// ---- GlobalTextList.TcGTLO
TEXTLIST GlobalTextList
  3955 = ' %5.2f h'
  1376 = ' %d %%'
  307 = ' %d days'
  1111 = '%2.1f  mA'
  102 = '%5.1f W'
  269 = '%5.2f h'
  621 = '%d'
  1617 = '%d %%'
  2081 = '%d days'
  3200 = '%d h'
  1372 = '%d Hz'
  2105 = '%d min'
  2025 = '%d ms'
  1540 = '%d s'
  1613 = '%d V'
  2272 = '%d weeks'
  1359 = '%d °C'
  376 = '%s'
  640 = '0'
  641 = '1'
  661 = '10'
  662 = '11'
  663 = '12'
  999 = '13'
  1000 = '14'
  1001 = '15'
  1002 = '16'
  1003 = '17'
  1004 = '18'
  1005 = '19'
  195 = '2'
  1006 = '20'
  1007 = '21'
  1008 = '22'
  1009 = '23'
  1010 = '24'
  1011 = '25'
  1012 = '26'
  1013 = '27'
  1014 = '28'
  1015 = '29'
  654 = '3'
  1016 = '30'
  1017 = '31'
  1018 = '32'
  1019 = '33'
  1020 = '34'
  1021 = '35'
  1022 = '36'
  1023 = '37'
  1024 = '38'
  1025 = '39'
  655 = '4'
  1026 = '40'
  1027 = '41'
  1028 = '42'
  1029 = '43'
  1030 = '44'
  1031 = '45'
  1032 = '46'
  1033 = '47'
  1034 = '48'
  1035 = '49'
  656 = '5'
  358 = '50'
  359 = '51'
  360 = '52'
  361 = '53'
  362 = '54'
  363 = '55'
  364 = '56'
  365 = '57'
  366 = '58'
  367 = '59'
  657 = '6'
  368 = '60'
  369 = '61'
  370 = '62'
  371 = '63'
  658 = '7'
  659 = '8'
  660 = '9'
  1089 = 'AC-supply possible'
  644 = 'Actual Level:'
  650 = 'Address Type'
  236 = 'Addressing Per Physical Selection Supported'
  1533 = 'Adjustable Emergency Level'
  1175 = 'AM Operation active:'
  1044 = 'AM operation possible'
  1045 = 'Auto Test Capability'
  1799 = 'Battery Charge'
  710 = 'Battery Duration Failure'
  3347 = 'Battery Failure'
  3316 = 'Battery Fully Charged'
  2471 = 'Bit 0'
  379 = 'Bit 1'
  2734 = 'Bit 2'
  2320 = 'Bit 3'
  929 = 'Bit 4'
  2576 = 'Bit 5'
  2065 = 'Bit 6'
  1623 = 'Bit 7'
  6 = 'Bottom Button'
  728 = 'Broadcast'
  482 = 'Button 1'
  720 = 'Button 2'
  515 = 'Button pressed'
  498 = 'Button released'
  527 = 'Button stuck / free'
  3304 = 'Cancel Hold Timer'
  2101 = 'Catch Movement'
  2319 = 'Catching:'
  897 = 'Change Addresses'
  1971 = 'Checkbox'
  372 = 'Choose group:'
  98 = 'Choose scene:'
  1571 = 'Circuit Failure'
  672 = 'Commands'
  618 = 'Complete new installation \n(all addresses will be removed)'
  807 = 'Control'
  645 = 'Control Gear Failure:'
  445 = 'Current protection active:'
  1716 = 'Current protection device'
  668 = 'Current protection enabled:'
  5 = 'Current Protector Enabled '
  1902 = 'DALI Line:'
  1135 = 'DC-supply possible'
  560 = 'Deadtime Timer:'
  1180 = 'DI1 falling edge'
  1218 = 'DI1 rising edge'
  1726 = 'DI2 falling edge'
  1876 = 'DI2 rising edge'
  519 = 'Dim Dwn'
  63 = 'Dim Up'
  2002 = 'Dimmer Temperature'
  936 = 'Dimming Curve:'
  1317 = 'Dimming method bit 0'
  776 = 'Dimming method bit 1'
  2135 = 'Do not lock process image in case of \nDALI commands from DI1 or DI2'
  4011 = 'Double press'
  1112 = 'Double Timer Min:'
  3936 = 'Double Timer:'
  811 = 'Down'
  594 = 'Down Switch-Off Threshold'
  2357 = 'Down Switch-On Threshold'
  1482 = 'Duration Test Delay Time'
  3527 = 'Duration Test Done And Result Valid'
  3086 = 'Duration Test Failed'
  3077 = 'Duration Test Interval'
  2631 = 'Duration Test Is In Progress'
  2791 = 'Duration Test Max. Delay Exceed'
  1708 = 'Duration Test Request Pending'
  2905 = 'Duration Test Result'
  1759 = 'Emergency Lamp Failure'
  779 = 'Emergency Level'
  3733 = 'Emergency MaxLevel'
  3168 = 'Emergency Min Level'
  1204 = 'Emergency Mode'
  971 = 'Emergency Mode Active'
  1901 = 'Emergency Status'
  486 = 'Enable'
  828 = 'Enable:'
  1982 = 'EventPriority'
  32 = 'EventPriority:'
  494 = 'EventScheme'
  1113 = 'EventScheme:'
  125 = 'Extended Emergency Mode Active'
  1841 = 'Extended Fade Time only valid if Fade Time equals 0!'
  3956 = 'Extended Version'
  649 = 'Fade Running:'
  1345 = 'FadeRate'
  1352 = 'FadeTime'
  1610 = 'Failure Status'
  319 = 'Fast Fade Time:'
  2099 = 'Features'
  425 = 'Features (Read only)'
  206 = 'Features Byte 1'
  377 = 'Features Byte 2'
  2876 = 'Features Byte 3'
  3334 = 'Function Test Delay Time'
  3242 = 'Function Test Done And Result Valid'
  2712 = 'Function Test Failed'
  1801 = 'Function Test Interval'
  1945 = 'Function Test Is In Progress'
  3448 = 'Function Test Max. Delay Exceed'
  165 = 'Function Test Request Pending'
  967 = 'Gang 1.312A'
  256 = 'Gang 1.315'
  906 = 'Gang 1.316'
  207 = 'Gang 2.344'
  66 = 'Gang 2.344A'
  406 = 'Gang 4.308'
  524 = 'Gang 6.310'
  316 = 'Gang 7.301'
  3204 = 'Gear Type'
  1989 = 'GearType'
  815 = 'Go to Scene'
  99 = 'Go to scene'
  721 = 'Group Address'
  2361 = 'Hardwired Inhibit Is Active'
  3553 = 'Hardwired Inhibit Supported'
  2225 = 'Hardwired Switch Is On'
  568 = 'Hold Timer:'
  199 = 'Hysteresis Min:'
  200 = 'Hysteresis:'
  790 = 'Identification Active'
  315 = 'Illuminance Level'
  37 = 'Inhibit'
  3340 = 'Inhibit Mode'
  540 = 'Input Value:'
  544 = 'Instance Error:'
  1038 = 'Instance Number:'
  3047 = 'Integral Control Gear'
  492 = 'Internal DALI power supply disabled'
  1771 = 'K-Bus Watchdog'
  3636 = 'Lamp Emergency Time'
  647 = 'Lamp Failure:'
  2812 = 'Lamp Total Operation Time'
  1521 = 'Leading Edge Mode Running'
  506 = 'LED module integrated'
  2077 = 'Linear Dimming Curve Active'
  2179 = 'Load current can be queried '
  1266 = 'Load Current Overload'
  1355 = 'Load current overload with output \nlevel reduction can be queried'
  306 = 'Load Decrease:'
  1137 = 'Load Increase:'
  2313 = 'Load over-current can be queried'
  2518 = 'Load Over-Current Shutdown'
  1226 = 'Load Rating'
  2963 = 'Load rating can be queried'
  2785 = 'Load unsuitable can be queried'
  1454 = 'Load voltage can be queried'
  516 = 'Load Voltage Out Of Limits'
  1811 = 'Lockable bytes: changeable if "Offset 2" has the Value 85 (0x55).\nFor changing use decimal value.'
  523 = 'Long press repeat'
  507 = 'Long press start'
  511 = 'Long press stop'
  43 = 'Lys Auto'
  444 = 'Lys Rum'
  489 = 'Lys Zone 1'
  2032 = 'Maintained Control Gear'
  2046 = 'Memory Bank:'
  3290 = 'Movement'
  531 = 'na'
  23 = 'Name'
  926 = 'Name of byte in memory bank'
  1417 = 'NewAddress'
  588 = 'No Movement'
  1061 = 'Non-logarithmic dimming curve can \nbe selected'
  1795 = 'Normal Mode Active'
  572 = 'Occupied'
  808 = 'Off'
  22 = 'Offset'
  1329 = 'Offset in memory bank'
  1409 = 'OldAddress'
  816 = 'On and Step Up'
  1207 = 'Open circuit detection can be queried'
  277 = 'Open Circuit:'
  1375 = 'Open Ciruit (No Load) Detect'
  619 = 'Optical feedback'
  963 = 'Output is current controlled'
  844 = 'Output regulated by current:'
  676 = 'Parameters'
  2547 = 'Parameters Absolute Input Device'
  1580 = 'Parameters Generic Instance'
  2259 = 'Parameters LED'
  309 = 'Parameters Light Sensor'
  556 = 'Parameters Occupancy Sensor'
  465 = 'Parameters Pushbutton Sensor'
  3234 = 'Physical Selection Supported'
  1847 = 'Physical selection supported'
  708 = 'PIR'
  457 = 'PIR status'
  1071 = 'Please check if Current Protector is present \nby reading parameters first.'
  308 = 'Please select the desired Short Address in the table above.'
  1458 = 'Please select the function you need from dropdown above'
  751 = 'Position Event'
  245 = 'Possible Operating Modes'
  719 = 'Power pulse operation'
  1744 = 'Power supply integrated'
  1561 = 'PP Operation active:'
  2321 = 'Prolong Time (30sec / Step)'
  970 = 'PWM Operation active:'
  1882 = 'PWM operation possible'
  1487 = 'Query idle time detection \nenabled'
  701 = 'Query load decrease enabled'
  1351 = 'Query load increase enabled'
  837 = 'Query reduction luminous flux \nregarding thermal overload'
  463 = 'Query short circuit enabled'
  1293 = 'Query thermal switch enabled'
  617 = 'Random Addressing'
  2174 = 'Rated Duration'
  881 = 'Re-Light / Reset Inhibit'
  373 = 'Read'
  1611 = 'Read Only'
  1531 = 'Reads all Fading Parameters'
  768 = 'Real Load Power'
  854 = 'Real load power can be queried'
  810 = 'Recall Max Level'
  809 = 'Recall Min Level'
  186 = 'Ref. Measurement failed:'
  439 = 'Reference System Power'
  2713 = 'Relight Rest Mode Supported'
  580 = 'Repeat'
  470 = 'Repeat Timer:'
  1913 = 'Report Timer:'
  716 = 'Reset Duration Test Done Flag'
  592 = 'Reset Function Test Done Flag'
  2418 = 'Reset inactive process image'
  3150 = 'Reset Lamp Time'
  648 = 'Reset State:'
  1037 = 'Resolution:'
  299 = 'Rest'
  591 = 'Rest Mode Active'
  2001 = 'RMS Load Current'
  784 = 'RMS Load Voltage'
  586 = 'RMS Supply Voltage'
  874 = 'Rum 1.106'
  65 = 'Rum 1.108'
  175 = 'Rum 1.111A'
  924 = 'Rum 1.111C'
  219 = 'Rum 1.111D'
  690 = 'Rum 1.111E'
  912 = 'Rum 1.115'
  126 = 'Rum 1.118'
  215 = 'Rum 1.312A'
  725 = 'Rum 1.318'
  839 = 'Rum 1.319'
  456 = 'Rum 1.320'
  800 = 'Rum 1.321'
  622 = 'Rum 1.322'
  646 = 'Rum 1.323'
  966 = 'Rum 1.324'
  95 = 'Rum 1.325'
  335 = 'Rum 1.326'
  150 = 'Rum 1.327'
  651 = 'Rum 1.328'
  980 = 'Rum 1.330'
  262 = 'Rum 1115'
  642 = 'Rum 2.341'
  978 = 'Rum 2.345'
  736 = 'Rum 2.349'
  430 = 'Rum 6.310 Sofagruppe'
  348 = 'Rum 6.327'
  891 = 'Rum 6.328'
  11 = 'Rum 6.329'
  72 = 'Rum 6.330B'
  197 = 'Rum 6.331'
  564 = 'Rum 6.333'
  997 = 'Rum 6.337'
  31 = 'Rum 6_330A'
  616 = 'Scan devices by address'
  1036 = 'Scene Level'
  814 = 'Scene:'
  1366 = 'Set Extended Fade Time'
  252 = 'Set Fade Rate'
  1875 = 'Set Fade Time'
  715 = 'Short Address'
  1367 = 'Short Address Range'
  1041 = 'Short Address:'
  34 = 'Short Circuit:'
  503 = 'Short press'
  1516 = 'Short Timer Min:'
  478 = 'Short Timer:'
  2548 = 'Shutdown Invalid Dimming Method'
  1360 = 'Single Short Address'
  395 = 'SP_Lux: %.0f'
  525 = 'SP_Lux: %f'
  615 = 'Start'
  582 = 'Start Duration Test'
  2374 = 'Start Function Test'
  155 = 'Start Identification'
  620 = 'Start with address:'
  2346 = 'State Incandescent Lamp'
  643 = 'Status'
  958 = 'Status Absolute Input Device'
  2506 = 'Status Generic Instance'
  2252 = 'Status LED'
  317 = 'Status Light Sensor'
  597 = 'Status Occupancy Sensor'
  536 = 'Status Pushbutton Sensor'
  558 = 'Step Down'
  813 = 'Step Down and Off'
  818 = 'Step Up'
  1193 = 'Stop Test'
  164 = 'Stuck Timer:'
  1256 = 'Supply Frequency'
  2271 = 'Supply frequency can be queried'
  1975 = 'Supply Frequency Out of Limits'
  2505 = 'Supply voltage can be queried'
  2707 = 'Supply Voltage Out Of Limits'
  1042 = 'Switch Off'
  375 = 'Switch On'
  3781 = 'Switched Maintained Control Gear'
  2168 = 'Temperature can be queried'
  2458 = 'Terminal Event'
  1848 = 'Test Execution Timeout'
  849 = 'Test Type A'
  2013 = 'Thermal Overload'
  2042 = 'Thermal Overload with output\nlevel reduction can be queried'
  1108 = 'Thermal Overload:'
  355 = 'Thermal Shut Down:'
  2507 = 'Thermal Shutdown'
  2226 = 'Thermal Shutdown can be queried'
  2733 = 'Threshold Editable'
  305 = 'To'
  973 = 'Top Button'
  136 = 'Trailing Edge ModeRunning'
  734 = 'Unaddressed'
  817 = 'Up'
  3123 = 'Up Switch-Off Threshold'
  1449 = 'Up Switch-On Threshold'
  2521 = 'V%s'
  576 = 'Vacant'
  1205 = 'Value'
  24 = 'Value Dec'
  1435 = 'Value decimal'
  25 = 'Value Hex'
  2231 = 'Value hexadecimal,\nto change use\nvalue decimal'
  374 = 'Write'
  2104 = 'Write\nDimming Curve'
  1047 = 'Write default values'
  490 = 'Write parameters'
END_TEXTLIST

// ---- POUs/Alle_Rum/Gange/Gang_1_316/Visualization_1_316.TcVIS
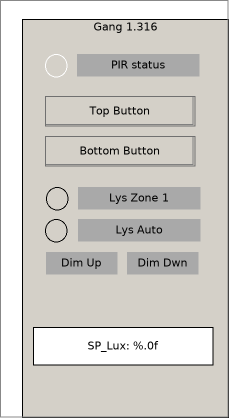
VISUALIZATION Visualization_1_316  // 229x418
    RoundedRectangle (22,19 207x399), "Gang 1.316"
    Rectangle (33,327 180x38), "SP_Lux: %.0f", text variable: P_Gang_1_316.fbLys.fbLightCtrl.fLuxZone1
    Button (45,96 150x30), "Top Button"
        tap P_Gang_1_316.bButtonZone1_Visu
    Button (45,136 150x30), "Bottom Button"
        tap P_Gang_1_316.bBottomButtonZone1_Visu
    Ellipse (46,187 22x23), colour toggle: P_Gang_1_316.fbLys.fbLightCtrl.bOnZone1
    Rectangle (78,187 122x22), "Lys Zone 1"
    Rectangle (46,252 71x22), "Dim Up", colour toggle: P_Gang_1_316.fbLys.fbLightCtrl.bDimUp
    Rectangle (127,252 71x22), "Dim Dwn", colour toggle: P_Gang_1_316.fbLys.fbLightCtrl.bDimDwn
    Ellipse (45,219 22x23), colour toggle: P_Gang_1_316.fbLys.fbLightCtrl.bAutoZone1
    Rectangle (78,219 122x22), "Lys Auto"
    Ellipse (45,54 22x23), colour toggle: P_Gang_1_316.fbLys.fbLightCtrl.bPIR
    Rectangle (77,54 122x22), "PIR status"
END_VISUALIZATION

// ---- POUs/Alle_Rum/Gange/Gang_7_301_en_linje_en_pendel_1/Visualization_4_308_1_1.TcVIS
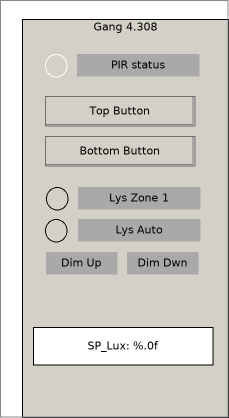
VISUALIZATION Visualization_4_308_1_1  // 229x418
    RoundedRectangle (22,19 207x399), "Gang 4.308"
    Rectangle (33,327 180x38), "SP_Lux: %.0f", text variable: P_Gang_4_308.arrfbLysGruppe[1].fbLightCtrl.fLuxZone1
    Button (45,96 150x30), "Top Button"
        tap P_Gang_4_308.bButtonZone1_Visu
    Button (45,136 150x30), "Bottom Button"
        tap P_Gang_4_308.bBottomButtonZone1_Visu
    Ellipse (46,187 22x23), colour toggle: P_Gang_4_308.fbLys.fbLightCtrl.bOnZone1
    Rectangle (78,187 122x22), "Lys Zone 1"
    Rectangle (46,252 71x22), "Dim Up", colour toggle: P_Gang_4_308.arrfbLysGruppe[1].fbLightCtrl.bDimUp
    Rectangle (127,252 71x22), "Dim Dwn", colour toggle: P_Gang_4_308.arrfbLysGruppe[1].fbLightCtrl.bDimDwn
    Ellipse (45,219 22x23), colour toggle: P_Gang_4_308.arrfbLysGruppe[1].fbLightCtrl.bAutoZone1
    Rectangle (78,219 122x22), "Lys Auto"
    Ellipse (45,54 22x23), colour toggle: P_Gang_4_308.arrfbLysGruppe[1].fbLightCtrl.bPIR
    Rectangle (77,54 122x22), "PIR status"
END_VISUALIZATION

// ---- POUs/Alle_Rum/Gange/Gang_2_346A/Visualization_2_346A.TcVIS
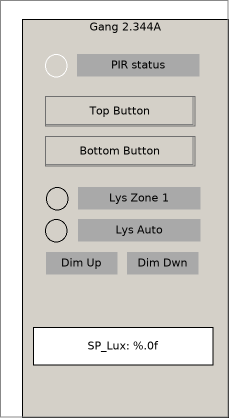
VISUALIZATION Visualization_2_346A  // 229x418
    RoundedRectangle (22,19 207x399), "Gang 2.344A"
    Rectangle (33,327 180x38), "SP_Lux: %.0f", text variable: P_Gang_2_346A.fbLys.fbLightCtrl.fLuxZone1
    Button (45,96 150x30), "Top Button"
        tap P_Gang_2_346A.bTopButtonZone1_Visu
    Button (45,136 150x30), "Bottom Button"
        tap P_Gang_2_346A.bBottomButtonZone1_Visu
    Ellipse (46,187 22x23), colour toggle: P_Gang_2_346A.fbLys.fbLightCtrl.bOnZone1
    Rectangle (78,187 122x22), "Lys Zone 1"
    Rectangle (46,252 71x22), "Dim Up", colour toggle: P_Gang_2_346A.fbLys.fbLightCtrl.bDimUp
    Rectangle (127,252 71x22), "Dim Dwn", colour toggle: P_Gang_2_346A.fbLys.fbLightCtrl.bDimDwn
    Ellipse (45,219 22x23), colour toggle: P_Gang_2_346A.fbLys.fbLightCtrl.bAutoZone1
    Rectangle (78,219 122x22), "Lys Auto"
    Ellipse (45,54 22x23), colour toggle: P_Gang_2_346A.fbLys.fbLightCtrl.bPIR
    Rectangle (77,54 122x22), "PIR status"
END_VISUALIZATION

// ---- POUs/Alle_Rum/Gange/Gang_2_344/Visualization_4_308_1_1_1.TcVIS
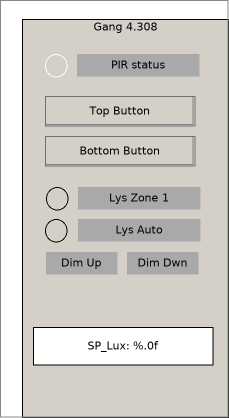
VISUALIZATION Visualization_4_308_1_1_1  // 229x418
    RoundedRectangle (22,19 207x399), "Gang 4.308"
    Rectangle (33,327 180x38), "SP_Lux: %.0f", text variable: P_Gang_4_308.arrfbLysGruppe[1].fbLightCtrl.fLuxZone1
    Button (45,96 150x30), "Top Button"
        tap P_Gang_4_308.bButtonZone1_Visu
    Button (45,136 150x30), "Bottom Button"
        tap P_Gang_4_308.bBottomButtonZone1_Visu
    Ellipse (46,187 22x23), colour toggle: P_Gang_4_308.fbLys.fbLightCtrl.bOnZone1
    Rectangle (78,187 122x22), "Lys Zone 1"
    Rectangle (46,252 71x22), "Dim Up", colour toggle: P_Gang_4_308.arrfbLysGruppe[1].fbLightCtrl.bDimUp
    Rectangle (127,252 71x22), "Dim Dwn", colour toggle: P_Gang_4_308.arrfbLysGruppe[1].fbLightCtrl.bDimDwn
    Ellipse (45,219 22x23), colour toggle: P_Gang_4_308.arrfbLysGruppe[1].fbLightCtrl.bAutoZone1
    Rectangle (78,219 122x22), "Lys Auto"
    Ellipse (45,54 22x23), colour toggle: P_Gang_4_308.arrfbLysGruppe[1].fbLightCtrl.bPIR
    Rectangle (77,54 122x22), "PIR status"
END_VISUALIZATION

// ---- POUs/Alle_Rum/Rum_Med_DALI_Pir/Rum_2_341/Visualization_2_341.TcVIS
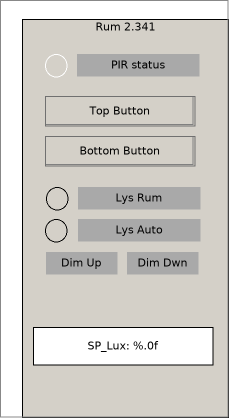
VISUALIZATION Visualization_2_341  // 229x418
    RoundedRectangle (22,19 207x399), "Rum 2.341"
    Rectangle (33,327 180x38), "SP_Lux: %.0f", text variable: P_Rum_2_341.fbLys.fbLightCtrl.fLuxZone1
    Button (45,96 150x30), "Top Button"
        tap P_Rum_2_341.bTopButtonZone1_Visu
    Button (45,136 150x30), "Bottom Button"
        tap P_Rum_2_341.bBottomButtonZone1_Visu
    Ellipse (46,187 22x23), colour toggle: P_Rum_2_341.fbLys.fbLightCtrl.bOnZone1
    Rectangle (78,187 122x22), "Lys Rum"
    Rectangle (46,252 71x22), "Dim Up", colour toggle: P_Rum_2_341.fbLys.fbLightCtrl.bDimUp
    Rectangle (127,252 71x22), "Dim Dwn", colour toggle: P_Rum_2_341.fbLys.fbLightCtrl.bDimDwn
    Ellipse (45,219 22x23), colour toggle: P_Rum_2_341.fbLys.fbLightCtrl.bAutoZone1
    Rectangle (78,219 122x22), "Lys Auto"
    Ellipse (45,54 22x23), colour toggle: P_Rum_2_341.fbLys.fbLightCtrl.bPIR
    Rectangle (77,54 122x22), "PIR status"
END_VISUALIZATION

// ---- POUs/Alle_Rum/Rum_Med_DALI_Pir/Rum_2_345/Visualization_2_345.TcVIS
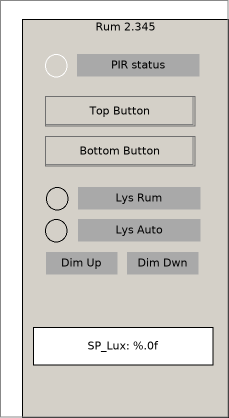
VISUALIZATION Visualization_2_345  // 229x418
    RoundedRectangle (22,19 207x399), "Rum 2.345"
    Rectangle (33,327 180x38), "SP_Lux: %.0f", text variable: P_Rum_2_345.fbLys.fbLightCtrl.fLuxZone1
    Button (45,96 150x30), "Top Button"
        tap P_Rum_2_345.bTopButtonZone1_Visu
    Button (45,136 150x30), "Bottom Button"
        tap P_Rum_2_345.bBottomButtonZone1_Visu
    Ellipse (46,187 22x23), colour toggle: P_Rum_2_345.fbLys.fbLightCtrl.bOnZone1
    Rectangle (78,187 122x22), "Lys Rum"
    Rectangle (46,252 71x22), "Dim Up", colour toggle: P_Rum_2_345.fbLys.fbLightCtrl.bDimUp
    Rectangle (127,252 71x22), "Dim Dwn", colour toggle: P_Rum_2_345.fbLys.fbLightCtrl.bDimDwn
    Ellipse (45,219 22x23), colour toggle: P_Rum_2_345.fbLys.fbLightCtrl.bAutoZone1
    Rectangle (78,219 122x22), "Lys Auto"
    Ellipse (45,54 22x23), colour toggle: P_Rum_2_345.fbLys.fbLightCtrl.bPIR
    Rectangle (77,54 122x22), "PIR status"
END_VISUALIZATION

// ---- POUs/Alle_Rum/Rum_Med_DALI_Pir/Rum_2_349/Visualization_2_349.TcVIS
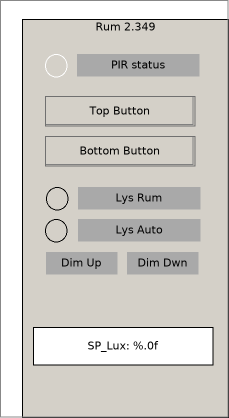
VISUALIZATION Visualization_2_349  // 229x418
    RoundedRectangle (22,19 207x399), "Rum 2.349"
    Rectangle (33,327 180x38), "SP_Lux: %.0f", text variable: P_Rum_2_349.fbLys.fbLightCtrl.fLuxZone1
    Button (45,96 150x30), "Top Button"
        tap P_Rum_2_349.bTopButtonZone1_Visu
    Button (45,136 150x30), "Bottom Button"
        tap P_Rum_2_349.bBottomButtonZone1_Visu
    Ellipse (46,187 22x23), colour toggle: P_Rum_2_349.fbLys.fbLightCtrl.bOnZone1
    Rectangle (78,187 122x22), "Lys Rum"
    Rectangle (46,252 71x22), "Dim Up", colour toggle: P_Rum_2_349.fbLys.fbLightCtrl.bDimUp
    Rectangle (127,252 71x22), "Dim Dwn", colour toggle: P_Rum_2_349.fbLys.fbLightCtrl.bDimDwn
    Ellipse (45,219 22x23), colour toggle: P_Rum_2_349.fbLys.fbLightCtrl.bAutoZone1
    Rectangle (78,219 122x22), "Lys Auto"
    Ellipse (45,54 22x23), colour toggle: P_Rum_2_349.fbLys.fbLightCtrl.bPIR
    Rectangle (77,54 122x22), "PIR status"
END_VISUALIZATION

// ---- POUs/DALI/DALI_Setup/VISUs/TextLists/CommandOnTerminalEvent.TcTLO
TEXTLIST CommandOnTerminalEvent
  0 = 'Do Nothing'
  1 = 'Off'
  2 = 'RecallMaxLevel'
  3 = 'RecallMinLevel'
  4 = 'GoToScene0'
  5 = 'GoToScene1'
  6 = 'GoToScene2'
  7 = 'GoToScene3'
  8 = 'GoToScene4'
  9 = 'GoToScene5'
  10 = 'GoToScene6'
  11 = 'GoToScene7'
  12 = 'GoToScene8'
  13 = 'GoToScene9'
  14 = 'GoToScene10'
  15 = 'GoToScene11'
  16 = 'GoToScene12'
  17 = 'GoToScene13'
  18 = 'GoToScene14'
  19 = 'GoToScene15'
   = ''
END_TEXTLIST

// ---- POUs/DALI/DALI_Setup/VISUs/TextLists/DimmingCurve.TcTLO
TEXTLIST DimmingCurve
  0 = 'Standard'
  1 = 'Linear'
  255 = 'Unknown'
   = ''
END_TEXTLIST

// ---- POUs/DALI/DALI_Setup/VISUs/TextLists/EventPriority.TcTLO
TEXTLIST EventPriority
  2 = 'MiddleHigh'
  3 = 'Middle'
  4 = 'MiddleLow'
  5 = 'Low'
  255 = 'Unknown'
   = ''
END_TEXTLIST

// ---- POUs/DALI/DALI_Setup/VISUs/TextLists/EventScheme.TcTLO
TEXTLIST EventScheme
  0 = '0 - Instance type and number'
  1 = '1 - Short address and instance type'
  2 = '2 - Short address and instance number'
  3 = '3 - Device group and instance type'
  4 = '4 - Instance group and instance type'
   = ''
END_TEXTLIST

// ---- POUs/DALI/DALI_Setup/VISUs/TextLists/ExtendedFadeTime.TcTLO
TEXTLIST ExtendedFadeTime
  0 = 'No Fade'
  1 = '1 * 100 ms = 100 ms'
  2 = '2 * 100 ms = 200 ms'
  3 = '3 * 100 ms = 300 ms'
  4 = '4 * 100 ms = 400 ms'
  5 = '5 * 100 ms = 500 ms'
  6 = '6 * 100 ms = 600 ms'
  7 = '7 * 100 ms = 700 ms'
  8 = '8 * 100 ms = 800 ms'
  9 = '9 * 100 ms = 900 ms'
  10 = '10 * 100 ms = 1000 ms'
  11 = '11 * 100 ms = 1100 ms'
  12 = '12 * 100 ms = 1200 ms'
  13 = '13 * 100 ms = 1300 ms'
  14 = '14 * 100 ms = 1400 ms'
  15 = '15 * 100 ms = 1500 ms'
  16 = '16 * 100 ms = 1600 ms'
  17 = '1 * 1 s = 1 s'
  18 = '2 * 1 s = 2 s'
  19 = '3 * 1 s = 3 s'
  20 = '4 * 1 s = 4 s'
  21 = '5 * 1 s = 5 s'
  22 = '6 * 1 s = 6 s'
  23 = '7 * 1 s = 7 s'
  24 = '8 * 1 s = 8 s'
  25 = '9 * 1 s = 9 s'
  26 = '10 * 1 s = 10 s'
  27 = '11 * 1 s = 11 s'
  28 = '12 * 1 s = 12 s'
  29 = '13 * 1 s = 13 s'
  30 = '14 * 1 s = 14 s'
  31 = '15 * 1 s = 15 s'
  32 = '16 * 1 s = 16 s'
  33 = '1 * 10 s = 10 s'
  34 = '2 * 10 s = 20 s'
  35 = '3 * 10 s = 30 s'
  36 = '4 * 10 s = 40 s'
  37 = '5 * 10 s = 50 s'
  38 = '6 * 10 s = 60 s'
  39 = '7 * 10 s = 70 s'
  40 = '8 * 10 s = 80 s'
  41 = '9 * 10 s = 90 s'
  42 = '10 * 10 s = 100 s'
  43 = '11 * 10 s = 110 s'
  44 = '12 * 10 s = 120 s'
  45 = '13 * 10 s = 130 s'
  46 = '14 * 10 s = 140 s'
  47 = '15 * 10 s = 150 s'
  48 = '16 * 10 s = 160 s'
  49 = '1 * 1 min = 1 min'
  50 = '2 * 1 min = 2 min'
  51 = '3 * 1 min = 3 min'
  52 = '4 * 1 min = 4 min'
  53 = '5 * 1 min = 5 min'
  54 = '6 * 1 min = 6 min'
  55 = '7 * 1 min = 7 min'
  56 = '8 * 1 min = 8 min'
  57 = '9 * 1 min = 9 min'
  58 = '10 * 1 min = 10 min'
  59 = '11 * 1 min = 11 min'
  60 = '12 * 1 min = 12 min'
  61 = '13 * 1 min = 13 min'
  62 = '14 * 1 min = 14 min'
  63 = '15 * 1 min = 15 min'
  64 = '16 * 1 min = 16 min'
  255 = 'Unknown'
   = ''
END_TEXTLIST

// ---- POUs/DALI/DALI_Setup/VISUs/TextLists/FadeRate.TcTLO
TEXTLIST FadeRate
  0 = 'Unknown'
  1 = '358 steps/s'
  2 = '253 steps/s'
  3 = '179 steps/s'
  4 = '127 steps/s'
  5 = '89,4 steps/s'
  6 = '63,3 steps/s'
  7 = '44,7 steps/s'
  8 = '31,6 steps/s'
  9 = '22,4 steps/s'
  10 = '15,8 steps/s'
  11 = '11,2 steps/s'
  12 = '7,9 steps/s'
  13 = '5,6 steps/s'
  14 = '4,0 steps/s'
  15 = '2,8 steps/s'
  255 = 'Unknown'
   = ''
END_TEXTLIST

// ---- POUs/DALI/DALI_Setup/VISUs/TextLists/FadeTime.TcTLO
TEXTLIST FadeTime
  0 = 'Extended Fade Time'
  1 = '0,7 s'
  2 = '1,0 s'
  3 = '1,4 s'
  4 = '2,0 s'
  5 = '2,8 s'
  6 = '4,0 s'
  7 = '5,7 s'
  8 = '8,0 s'
  9 = '11,3 s'
  10 = '16,0 s'
  11 = '22,6 s'
  12 = '32,0 s'
  13 = '45,3 s'
  14 = '64,0 s'
  15 = '90,5 s'
   = ''
END_TEXTLIST

// ---- POUs/DALI/DALI_Setup/VISUs/TextLists/FastFadeTime.TcTLO
TEXTLIST FastFadeTime
  0 = 'Disabled'
  4 = 'T100ms'
  8 = 'T200ms'
  12 = 'T300ms'
  16 = 'T400ms'
  20 = 'T500ms'
  24 = 'T600ms'
  27 = 'T700ms'
  255 = 'Unknown'
   = ''
END_TEXTLIST

// ---- POUs/DALI/DALI_Setup/VISUs/TextLists/TextList_Dialogs.TcTLO
TEXTLIST TextList_Dialogs
  0 = 'Select the function'
  1 = 'Control Gears - Commands'
  2 = 'Control Gears - Addressing'
  3 = 'Control Gears - Parameters'
  4 = 'Control Gears - Groups'
  5 = 'Control Gears - Scenes'
  6 = 'Control Gears - Memory Pages'
  7 = 'Control Gears - Set Fading'
  8 = 'Control Gears - Device Type 1 (Emergency lighting)'
  9 = 'Control Gears - Device Type 4 (Incandescent lamp)'
  10 = 'Control Gears - Device Type 6 (LED)'
  11 = 'Control Gears - Device Type 7 (Switching)'
  12 = 'Control Devices - Addressing'
  13 = 'Control Devices - Parameters'
  15 = 'Control Devices - Device Type 1 (Push button)'
  16 = 'Control Devices - Device Type 2 (Absolute input)'
  17 = 'Control Devices - Device Type 3 (Occupancy sensor)'
  18 = 'Control Devices - Device Type 4 (Light sensor)'
  19 = 'Control Devices - Device Type 0 (Generic instance)'
  20 = 'Control Devices - Memory Pages'
  14 = 'Control Devices - Identify'
   = ''
END_TEXTLIST

// ---- POUs/DALI/DALI_Setup/VISUs/Visu_DALICommissioning/Visu_KL6821Configuration.TcVIS
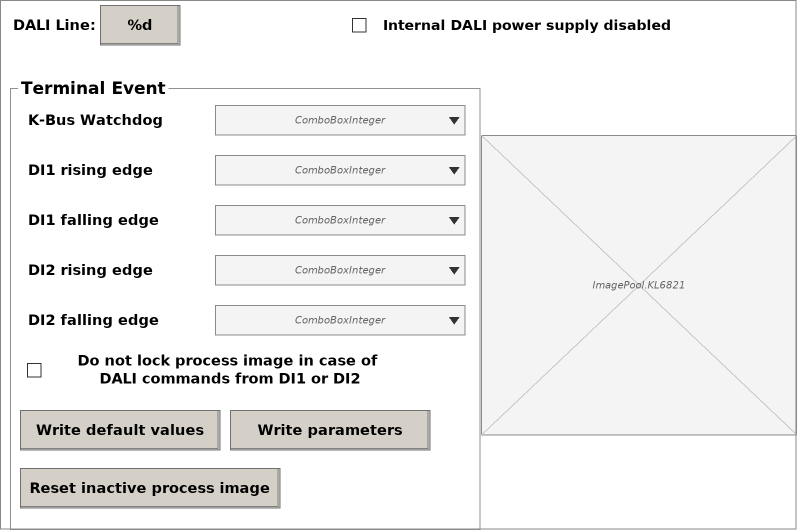
VISUALIZATION Visu_KL6821Configuration  // 797x530
    GroupBox (10,80 470x450), "Terminal Event"
        Textfield (15,25 170x30), "K-Bus Watchdog"
        ComboBoxInteger (205,25 250x30), variable: P_DALI_Background.eCommandKBusWatchdog, text list: 'CommandOnTerminalEvent'
        Textfield (15,75 170x30), "DI1 rising edge"
        Textfield (15,125 170x30), "DI1 falling edge"
        ComboBoxInteger (205,75 250x30), variable: P_DALI_Background.eCommandDI1RisingEdge, text list: 'CommandOnTerminalEvent'
        ComboBoxInteger (205,125 250x30), variable: P_DALI_Background.eCommandDI1FallingEdge, text list: 'CommandOnTerminalEvent'
        Textfield (15,175 170x30), "DI2 rising edge"
        ComboBoxInteger (205,175 250x30), variable: P_DALI_Background.eCommandDI2RisingEdge, text list: 'CommandOnTerminalEvent'
        Textfield (15,225 170x30), "DI2 falling edge"
        ComboBoxInteger (205,225 250x30), variable: P_DALI_Background.eCommandDI2FallingEdge, text list: 'CommandOnTerminalEvent'
        Button (220,330 200x40), "Write parameters"
            OnMouseClick: execute { P_DALI_Background.bInitialize := TRUE; }
        Button (10,330 200x40), "Write default values"
            OnMouseClick: execute { P_DALI_Background.bDefaultValues := TRUE; }
        Button (10,388 260x40), "Reset inactive process image"
            OnMouseClick: execute { P_DALI_Background.bResetInactiveProcessImage := TRUE; }
        Checkbox (15,275 35x30), variable: P_DALI_Background.bDoNotLockProcessImage
        Textfield (50,267 340x45), "Do not lock process image in case of DALI commands from DI1 or DI2"
    Image (481,135 316x300), image: ImagePool.KL6821
    Group (350,10 330x30)
        Checkbox (0,0 34x30), variable: P_DALI_Background.bInternalPowerSupplyDisabled
        Textfield (30,0 294x30), "Internal DALI power supply disabled"
    Group (10,5 170x40)
        Textfield (0,0 110x40), "DALI Line:"
        Button (90,0 80x40), "%d", text variable: GVL_Internal.nDALILine
            OnMouseClick: write the text variable via Default, min 1, max 10, title "Choose line"
END_VISUALIZATION

// ---- POUs/DALI/DALI_Setup/VISUs/Visu_DALICommissioning/Visu_Part102Commands.TcVIS
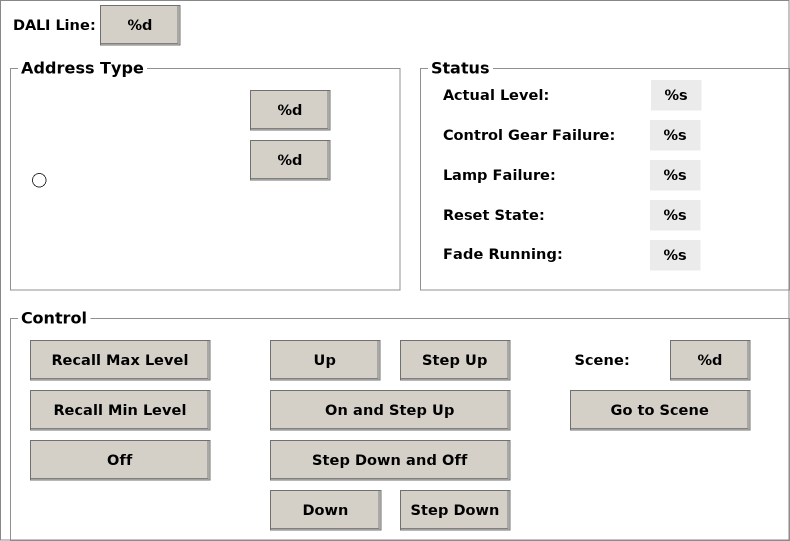
VISUALIZATION Visu_Part102Commands  // 790x541
    GroupBox (10,310 780x231), "Control"
        Button (20,130 180x40), "Off"
            OnMouseClick: execute { DALI_Commissioning.fbPart102Commands.bOff := TRUE; }
        Button (20,80 180x40), "Recall Min Level"
            OnMouseClick: execute { DALI_Commissioning.fbPart102Commands.bRecallMinLevel := TRUE; }
        Button (20,30 180x40), "Recall Max Level"
            OnMouseClick: execute { DALI_Commissioning.fbPart102Commands.bRecallMaxLevel := TRUE; }
        Button (260,180 111x40), "Down"
            OnMouseClick: execute { DALI_Commissioning.fbPart102Commands.bDown := TRUE; }
        Button (390,180 110x40), "Step Down"
            OnMouseClick: execute { DALI_Commissioning.fbPart102Commands.bStepDown := TRUE; }
        Button (260,130 240x40), "Step Down and Off"
            OnMouseClick: execute { DALI_Commissioning.fbPart102Commands.bStepDownAndOff := TRUE; }
        Button (660,30 80x40), "%d", text variable: DALI_Commissioning.fbPart102Commands.nScene
            OnMouseClick: write the text variable via Default, min 0, max 15, title "Insert scene number"
        Textfield (550,35 85x30), "Scene:"
        Button (560,80 180x40), "Go to Scene"
            OnMouseClick: execute { DALI_Commissioning.fbPart102Commands.bGotoScene := TRUE; }
        Button (260,80 240x40), "On and Step Up"
            OnMouseClick: execute { DALI_Commissioning.fbPart102Commands.bOnAndStepUp := TRUE; }
        Button (260,30 110x40), "Up"
            OnMouseClick: execute { DALI_Commissioning.fbPart102Commands.bUp := TRUE; }
        Button (390,30 110x40), "Step Up"
            OnMouseClick: execute { DALI_Commissioning.fbPart102Commands.bStepUp := TRUE; }
    GroupBox (420,60 370x230), "Status"
        Textfield (20,20 200x30), "Actual Level:"
        Textfield (20,60 200x30), "Control Gear Failure:"
        Textfield (231,20 50x30), "%s", text variable: DALI_Commissioning.fbPart102Commands.sActualLevel
        Textfield (230,60 50x30), "%s", text variable: DALI_Commissioning.fbPart102Commands.sControlGearFailure
        Textfield (20,100 200x30), "Lamp Failure:"
        Textfield (230,100 50x30), "%s", text variable: DALI_Commissioning.fbPart102Commands.sLampFailure
        Textfield (20,140 200x30), "Reset State:"
        Textfield (230,140 50x30), "%s", text variable: DALI_Commissioning.fbPart102Commands.sResetState
        Textfield (20,180 200x28), "Fade Running:"
        Textfield (230,180 50x30), "%s", text variable: DALI_Commissioning.fbPart102Commands.sFadeRunning
    GroupBox (10,60 390x230), "Address Type"
        Button (240,30 80x40), "%d", text variable: DALI_Commissioning.fbPart102Commands.nShortAddress
            OnMouseClick: write the text variable via Default, min 0, max 63, title "Insert Short Address"
            OnMouseClick: execute {  }
        RadioButton (20,20 190x200), variable: DALI_Commissioning.fbPart102Commands.eAddressType
            Areas[0]: Text=Short Address
            Areas[1]: Text=Group Address
            Areas[2]: Text=Broadcast
            Areas[3]: Text=Unaddressed
        Button (240,80 80x40), "%d", text variable: DALI_Commissioning.fbPart102Commands.nGroupAddress
            OnMouseClick: write the text variable via Default, min 0, max 15, title "Insert Group Address"
    Group (10,5 170x40)
        Textfield (0,0 110x40), "DALI Line:"
        Button (90,0 80x40), "%d", text variable: GVL_Internal.nDALILine
            OnMouseClick: write the text variable via Default, min 1, max 10, title "Choose line"
END_VISUALIZATION

// ---- POUs/DALI/DALI_Setup/VISUs/Visu_DALICommissioning/Visu_Part102Groups.TcVIS
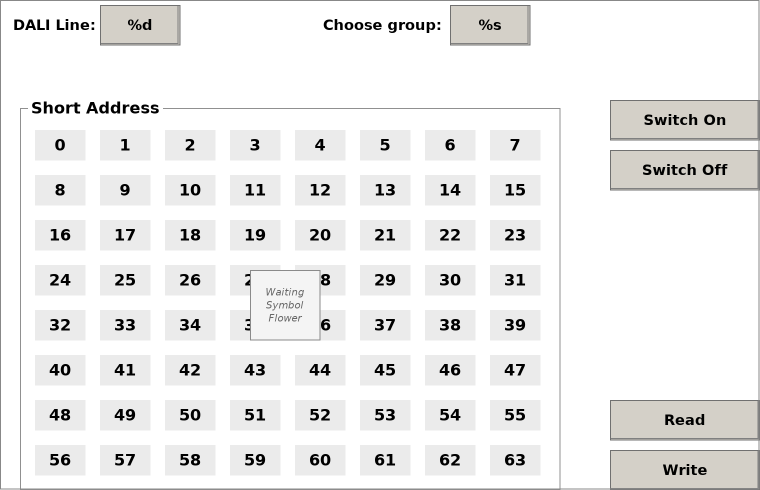
VISUALIZATION Visu_Part102Groups  // 760x490
    GroupBox (20,100 540x390), "Short Address"
        Textfield (15,30 50x30), "0", colour toggle: DALI_Commissioning.fbPart102Groups.aShowAlarmState[0] = TRUE, invisible if: DALI_Commissioning.fbPart102Groups.aActivateButton[0] = FALSE, input disabled if: DALI_Commissioning.fbPart102Groups.aActivateButton[0] = FALSE
            OnMouseClick: execute { DALI_Commissioning.fbPart102Groups.aButtonClick[0] := TRUE; }
        Textfield (80,30 50x30), "1", colour toggle: DALI_Commissioning.fbPart102Groups.aShowAlarmState[1] = TRUE, invisible if: DALI_Commissioning.fbPart102Groups.aActivateButton[1] = FALSE, input disabled if: DALI_Commissioning.fbPart102Groups.aActivateButton[1] = FALSE
            OnMouseClick: execute { DALI_Commissioning.fbPart102Groups.aButtonClick[1] := TRUE; }
        Textfield (145,30 50x30), "2", colour toggle: DALI_Commissioning.fbPart102Groups.aShowAlarmState[2] = TRUE, invisible if: DALI_Commissioning.fbPart102Groups.aActivateButton[2] = FALSE, input disabled if: DALI_Commissioning.fbPart102Groups.aActivateButton[2] = FALSE
            OnMouseClick: execute { DALI_Commissioning.fbPart102Groups.aButtonClick[2] := TRUE; }
        Textfield (210,30 50x30), "3", colour toggle: DALI_Commissioning.fbPart102Groups.aShowAlarmState[3] = TRUE, invisible if: DALI_Commissioning.fbPart102Groups.aActivateButton[3] = FALSE, input disabled if: DALI_Commissioning.fbPart102Groups.aActivateButton[3] = FALSE
            OnMouseClick: execute { DALI_Commissioning.fbPart102Groups.aButtonClick[3] := TRUE; }
        Textfield (275,30 50x30), "4", colour toggle: DALI_Commissioning.fbPart102Groups.aShowAlarmState[4] = TRUE, invisible if: DALI_Commissioning.fbPart102Groups.aActivateButton[4] = FALSE, input disabled if: DALI_Commissioning.fbPart102Groups.aActivateButton[4] = FALSE
            OnMouseClick: execute { DALI_Commissioning.fbPart102Groups.aButtonClick[4] := TRUE; }
        Textfield (340,30 50x30), "5", colour toggle: DALI_Commissioning.fbPart102Groups.aShowAlarmState[5] = TRUE, invisible if: DALI_Commissioning.fbPart102Groups.aActivateButton[5] = FALSE, input disabled if: DALI_Commissioning.fbPart102Groups.aActivateButton[5] = FALSE
            OnMouseClick: execute { DALI_Commissioning.fbPart102Groups.aButtonClick[5] := TRUE; }
        Textfield (405,30 50x30), "6", colour toggle: DALI_Commissioning.fbPart102Groups.aShowAlarmState[6] = TRUE, invisible if: DALI_Commissioning.fbPart102Groups.aActivateButton[6] = FALSE, input disabled if: DALI_Commissioning.fbPart102Groups.aActivateButton[6] = FALSE
            OnMouseClick: execute { DALI_Commissioning.fbPart102Groups.aButtonClick[6] := TRUE; }
        Textfield (470,30 50x30), "7", colour toggle: DALI_Commissioning.fbPart102Groups.aShowAlarmState[7] = TRUE, invisible if: DALI_Commissioning.fbPart102Groups.aActivateButton[7] = FALSE, input disabled if: DALI_Commissioning.fbPart102Groups.aActivateButton[7] = FALSE
            OnMouseClick: execute { DALI_Commissioning.fbPart102Groups.aButtonClick[7] := TRUE; }
        Textfield (15,75 50x30), "8", colour toggle: DALI_Commissioning.fbPart102Groups.aShowAlarmState[8] = TRUE, invisible if: DALI_Commissioning.fbPart102Groups.aActivateButton[8] = FALSE, input disabled if: DALI_Commissioning.fbPart102Groups.aActivateButton[8] = FALSE
            OnMouseClick: execute { DALI_Commissioning.fbPart102Groups.aButtonClick[8] := TRUE; }
        Textfield (80,75 50x30), "9", colour toggle: DALI_Commissioning.fbPart102Groups.aShowAlarmState[9] = TRUE, invisible if: DALI_Commissioning.fbPart102Groups.aActivateButton[9] = FALSE, input disabled if: DALI_Commissioning.fbPart102Groups.aActivateButton[9] = FALSE
            OnMouseClick: execute { DALI_Commissioning.fbPart102Groups.aButtonClick[9] := TRUE; }
        Textfield (145,75 50x30), "10", colour toggle: DALI_Commissioning.fbPart102Groups.aShowAlarmState[10] = TRUE, invisible if: DALI_Commissioning.fbPart102Groups.aActivateButton[10] = FALSE, input disabled if: DALI_Commissioning.fbPart102Groups.aActivateButton[10] = FALSE
            OnMouseClick: execute { DALI_Commissioning.fbPart102Groups.aButtonClick[10] := TRUE; }
        Textfield (210,75 50x30), "11", colour toggle: DALI_Commissioning.fbPart102Groups.aShowAlarmState[11] = TRUE, invisible if: DALI_Commissioning.fbPart102Groups.aActivateButton[11] = FALSE, input disabled if: DALI_Commissioning.fbPart102Groups.aActivateButton[11] = FALSE
            OnMouseClick: execute { DALI_Commissioning.fbPart102Groups.aButtonClick[11] := TRUE; }
        Textfield (275,75 50x30), "12", colour toggle: DALI_Commissioning.fbPart102Groups.aShowAlarmState[12] = TRUE, invisible if: DALI_Commissioning.fbPart102Groups.aActivateButton[12] = FALSE, input disabled if: DALI_Commissioning.fbPart102Groups.aActivateButton[12] = FALSE
            OnMouseClick: execute { DALI_Commissioning.fbPart102Groups.aButtonClick[12] := TRUE; }
        Textfield (340,75 50x30), "13", colour toggle: DALI_Commissioning.fbPart102Groups.aShowAlarmState[13] = TRUE, invisible if: DALI_Commissioning.fbPart102Groups.aActivateButton[13] = FALSE, input disabled if: DALI_Commissioning.fbPart102Groups.aActivateButton[13] = FALSE
            OnMouseClick: execute { DALI_Commissioning.fbPart102Groups.aButtonClick[13] := TRUE; }
        Textfield (405,75 50x30), "14", colour toggle: DALI_Commissioning.fbPart102Groups.aShowAlarmState[14] = TRUE, invisible if: DALI_Commissioning.fbPart102Groups.aActivateButton[14] = FALSE, input disabled if: DALI_Commissioning.fbPart102Groups.aActivateButton[14] = FALSE
            OnMouseClick: execute { DALI_Commissioning.fbPart102Groups.aButtonClick[14] := TRUE; }
        Textfield (470,75 50x30), "15", colour toggle: DALI_Commissioning.fbPart102Groups.aShowAlarmState[15] = TRUE, invisible if: DALI_Commissioning.fbPart102Groups.aActivateButton[15] = FALSE, input disabled if: DALI_Commissioning.fbPart102Groups.aActivateButton[15] = FALSE
            OnMouseClick: execute { DALI_Commissioning.fbPart102Groups.aButtonClick[15] := TRUE; }
        Textfield (15,120 50x30), "16", colour toggle: DALI_Commissioning.fbPart102Groups.aShowAlarmState[16] = TRUE, invisible if: DALI_Commissioning.fbPart102Groups.aActivateButton[16] = FALSE, input disabled if: DALI_Commissioning.fbPart102Groups.aActivateButton[16] = FALSE
            OnMouseClick: execute { DALI_Commissioning.fbPart102Groups.aButtonClick[16] := TRUE; }
        Textfield (80,120 50x30), "17", colour toggle: DALI_Commissioning.fbPart102Groups.aShowAlarmState[17] = TRUE, invisible if: DALI_Commissioning.fbPart102Groups.aActivateButton[17] = FALSE, input disabled if: DALI_Commissioning.fbPart102Groups.aActivateButton[17] = FALSE
            OnMouseClick: execute { DALI_Commissioning.fbPart102Groups.aButtonClick[17] := TRUE; }
        Textfield (145,120 50x30), "18", colour toggle: DALI_Commissioning.fbPart102Groups.aShowAlarmState[18] = TRUE, invisible if: DALI_Commissioning.fbPart102Groups.aActivateButton[18] = FALSE, input disabled if: DALI_Commissioning.fbPart102Groups.aActivateButton[18] = FALSE
            OnMouseClick: execute { DALI_Commissioning.fbPart102Groups.aButtonClick[18] := TRUE; }
        Textfield (210,120 50x30), "19", colour toggle: DALI_Commissioning.fbPart102Groups.aShowAlarmState[19] = TRUE, invisible if: DALI_Commissioning.fbPart102Groups.aActivateButton[19] = FALSE, input disabled if: DALI_Commissioning.fbPart102Groups.aActivateButton[19] = FALSE
            OnMouseClick: execute { DALI_Commissioning.fbPart102Groups.aButtonClick[19] := TRUE; }
        Textfield (275,120 50x30), "20", colour toggle: DALI_Commissioning.fbPart102Groups.aShowAlarmState[20] = TRUE, invisible if: DALI_Commissioning.fbPart102Groups.aActivateButton[20] = FALSE, input disabled if: DALI_Commissioning.fbPart102Groups.aActivateButton[20] = FALSE
            OnMouseClick: execute { DALI_Commissioning.fbPart102Groups.aButtonClick[20] := TRUE; }
        Textfield (340,120 50x30), "21", colour toggle: DALI_Commissioning.fbPart102Groups.aShowAlarmState[21] = TRUE, invisible if: DALI_Commissioning.fbPart102Groups.aActivateButton[21] = FALSE, input disabled if: DALI_Commissioning.fbPart102Groups.aActivateButton[21] = FALSE
            OnMouseClick: execute { DALI_Commissioning.fbPart102Groups.aButtonClick[21] := TRUE; }
        Textfield (405,120 50x30), "22", colour toggle: DALI_Commissioning.fbPart102Groups.aShowAlarmState[22] = TRUE, invisible if: DALI_Commissioning.fbPart102Groups.aActivateButton[22] = FALSE, input disabled if: DALI_Commissioning.fbPart102Groups.aActivateButton[22] = FALSE
            OnMouseClick: execute { DALI_Commissioning.fbPart102Groups.aButtonClick[22] := TRUE; }
        Textfield (470,120 50x30), "23", colour toggle: DALI_Commissioning.fbPart102Groups.aShowAlarmState[23] = TRUE, invisible if: DALI_Commissioning.fbPart102Groups.aActivateButton[23] = FALSE, input disabled if: DALI_Commissioning.fbPart102Groups.aActivateButton[23] = FALSE
            OnMouseClick: execute { DALI_Commissioning.fbPart102Groups.aButtonClick[23] := TRUE; }
        Textfield (15,165 50x30), "24", colour toggle: DALI_Commissioning.fbPart102Groups.aShowAlarmState[24] = TRUE, invisible if: DALI_Commissioning.fbPart102Groups.aDeviceGroupState[24] = 0, input disabled if: DALI_Commissioning.fbPart102Groups.aDeviceGroupState[24] = 0
            OnMouseClick: execute { DALI_Commissioning.fbPart102Groups.aButtonClick[24] := TRUE; }
        Textfield (80,165 50x30), "25", colour toggle: DALI_Commissioning.fbPart102Groups.aShowAlarmState[25] = TRUE, invisible if: DALI_Commissioning.fbPart102Groups.aActivateButton[25] = FALSE, input disabled if: DALI_Commissioning.fbPart102Groups.aActivateButton[25] = FALSE
            OnMouseClick: execute { DALI_Commissioning.fbPart102Groups.aButtonClick[25] := TRUE; }
        Textfield (145,165 50x30), "26", colour toggle: DALI_Commissioning.fbPart102Groups.aShowAlarmState[26] = TRUE, invisible if: DALI_Commissioning.fbPart102Groups.aActivateButton[26] = FALSE, input disabled if: DALI_Commissioning.fbPart102Groups.aActivateButton[26] = FALSE
            OnMouseClick: execute { DALI_Commissioning.fbPart102Groups.aButtonClick[26] := TRUE; }
        Textfield (210,165 50x30), "27", colour toggle: DALI_Commissioning.fbPart102Groups.aShowAlarmState[27] = TRUE, invisible if: DALI_Commissioning.fbPart102Groups.aActivateButton[27] = FALSE, input disabled if: DALI_Commissioning.fbPart102Groups.aActivateButton[27] = FALSE
            OnMouseClick: execute { DALI_Commissioning.fbPart102Groups.aButtonClick[27] := TRUE; }
        Textfield (275,165 50x30), "28", colour toggle: DALI_Commissioning.fbPart102Groups.aShowAlarmState[28] = TRUE, invisible if: DALI_Commissioning.fbPart102Groups.aActivateButton[28] = FALSE, input disabled if: DALI_Commissioning.fbPart102Groups.aActivateButton[28] = FALSE
            OnMouseClick: execute { DALI_Commissioning.fbPart102Groups.aButtonClick[28] := TRUE; }
        Textfield (340,165 50x30), "29", colour toggle: DALI_Commissioning.fbPart102Groups.aShowAlarmState[29] = TRUE, invisible if: DALI_Commissioning.fbPart102Groups.aActivateButton[29] = FALSE, input disabled if: DALI_Commissioning.fbPart102Groups.aActivateButton[29] = FALSE
            OnMouseClick: execute { DALI_Commissioning.fbPart102Groups.aButtonClick[29] := TRUE; }
        Textfield (405,165 50x30), "30", colour toggle: DALI_Commissioning.fbPart102Groups.aShowAlarmState[30] = TRUE, invisible if: DALI_Commissioning.fbPart102Groups.aActivateButton[30] = FALSE, input disabled if: DALI_Commissioning.fbPart102Groups.aActivateButton[30] = FALSE
            OnMouseClick: execute { DALI_Commissioning.fbPart102Groups.aButtonClick[30] := TRUE; }
        Textfield (470,165 50x30), "31", colour toggle: DALI_Commissioning.fbPart102Groups.aShowAlarmState[31] = TRUE, invisible if: DALI_Commissioning.fbPart102Groups.aActivateButton[31] = FALSE, input disabled if: DALI_Commissioning.fbPart102Groups.aActivateButton[31] = FALSE
            OnMouseClick: execute { DALI_Commissioning.fbPart102Groups.aButtonClick[31] := TRUE; }
        Textfield (15,210 50x30), "32", colour toggle: DALI_Commissioning.fbPart102Groups.aShowAlarmState[32] = TRUE, invisible if: DALI_Commissioning.fbPart102Groups.aActivateButton[32] = FALSE, input disabled if: DALI_Commissioning.fbPart102Groups.aActivateButton[32] = FALSE
            OnMouseClick: execute { DALI_Commissioning.fbPart102Groups.aButtonClick[32] := TRUE; }
        Textfield (80,210 50x30), "33", colour toggle: DALI_Commissioning.fbPart102Groups.aShowAlarmState[33] = TRUE, invisible if: DALI_Commissioning.fbPart102Groups.aActivateButton[33] = FALSE, input disabled if: DALI_Commissioning.fbPart102Groups.aActivateButton[33] = FALSE
            OnMouseClick: execute { DALI_Commissioning.fbPart102Groups.aButtonClick[33] := TRUE; }
        Textfield (145,210 50x30), "34", colour toggle: DALI_Commissioning.fbPart102Groups.aShowAlarmState[34] = TRUE, invisible if: DALI_Commissioning.fbPart102Groups.aActivateButton[34] = FALSE, input disabled if: DALI_Commissioning.fbPart102Groups.aActivateButton[34] = FALSE
            OnMouseClick: execute { DALI_Commissioning.fbPart102Groups.aButtonClick[34] := TRUE; }
        Textfield (210,210 50x30), "35", colour toggle: DALI_Commissioning.fbPart102Groups.aShowAlarmState[35] = TRUE, invisible if: DALI_Commissioning.fbPart102Groups.aActivateButton[35] = FALSE, input disabled if: DALI_Commissioning.fbPart102Groups.aActivateButton[35] = FALSE
            OnMouseClick: execute { DALI_Commissioning.fbPart102Groups.aButtonClick[35] := TRUE; }
        Textfield (275,210 50x30), "36", colour toggle: DALI_Commissioning.fbPart102Groups.aShowAlarmState[36] = TRUE, invisible if: DALI_Commissioning.fbPart102Groups.aActivateButton[36] = FALSE, input disabled if: DALI_Commissioning.fbPart102Groups.aActivateButton[36] = FALSE
            OnMouseClick: execute { DALI_Commissioning.fbPart102Groups.aButtonClick[36] := TRUE; }
        Textfield (340,210 50x30), "37", colour toggle: DALI_Commissioning.fbPart102Groups.aShowAlarmState[37] = TRUE, invisible if: DALI_Commissioning.fbPart102Groups.aActivateButton[37] = FALSE, input disabled if: DALI_Commissioning.fbPart102Groups.aActivateButton[37] = FALSE
            OnMouseClick: execute { DALI_Commissioning.fbPart102Groups.aButtonClick[37] := TRUE; }
        Textfield (405,210 50x30), "38", colour toggle: DALI_Commissioning.fbPart102Groups.aShowAlarmState[38] = TRUE, invisible if: DALI_Commissioning.fbPart102Groups.aActivateButton[38] = FALSE, input disabled if: DALI_Commissioning.fbPart102Groups.aActivateButton[38] = FALSE
            OnMouseClick: execute { DALI_Commissioning.fbPart102Groups.aButtonClick[38] := TRUE; }
        Textfield (470,210 50x30), "39", colour toggle: DALI_Commissioning.fbPart102Groups.aShowAlarmState[39] = TRUE, invisible if: DALI_Commissioning.fbPart102Groups.aActivateButton[39] = FALSE, input disabled if: DALI_Commissioning.fbPart102Groups.aActivateButton[39] = FALSE
            OnMouseClick: execute { DALI_Commissioning.fbPart102Groups.aButtonClick[39] := TRUE; }
        Textfield (15,255 50x30), "40", colour toggle: DALI_Commissioning.fbPart102Groups.aShowAlarmState[40] = TRUE, invisible if: DALI_Commissioning.fbPart102Groups.aActivateButton[40] = FALSE, input disabled if: DALI_Commissioning.fbPart102Groups.aActivateButton[40] = FALSE
            OnMouseClick: execute { DALI_Commissioning.fbPart102Groups.aButtonClick[40] := TRUE; }
        Textfield (80,255 50x30), "41", colour toggle: DALI_Commissioning.fbPart102Groups.aShowAlarmState[41] = TRUE, invisible if: DALI_Commissioning.fbPart102Groups.aActivateButton[41] = FALSE, input disabled if: DALI_Commissioning.fbPart102Groups.aActivateButton[41] = FALSE
            OnMouseClick: execute { DALI_Commissioning.fbPart102Groups.aButtonClick[41] := TRUE; }
        Textfield (145,255 50x30), "42", colour toggle: DALI_Commissioning.fbPart102Groups.aShowAlarmState[42] = TRUE, invisible if: DALI_Commissioning.fbPart102Groups.aActivateButton[42] = FALSE, input disabled if: DALI_Commissioning.fbPart102Groups.aActivateButton[42] = FALSE
            OnMouseClick: execute { DALI_Commissioning.fbPart102Groups.aButtonClick[42] := TRUE; }
        Textfield (210,255 50x30), "43", colour toggle: DALI_Commissioning.fbPart102Groups.aShowAlarmState[43] = TRUE, invisible if: DALI_Commissioning.fbPart102Groups.aActivateButton[43] = FALSE, input disabled if: DALI_Commissioning.fbPart102Groups.aActivateButton[43] = FALSE
            OnMouseClick: execute { DALI_Commissioning.fbPart102Groups.aButtonClick[43] := TRUE; }
        Textfield (275,255 50x30), "44", colour toggle: DALI_Commissioning.fbPart102Groups.aShowAlarmState[44] = TRUE, invisible if: DALI_Commissioning.fbPart102Groups.aActivateButton[44] = FALSE, input disabled if: DALI_Commissioning.fbPart102Groups.aActivateButton[44] = FALSE
            OnMouseClick: execute { DALI_Commissioning.fbPart102Groups.aButtonClick[44] := TRUE; }
        Textfield (340,255 50x30), "45", colour toggle: DALI_Commissioning.fbPart102Groups.aShowAlarmState[45] = TRUE, invisible if: DALI_Commissioning.fbPart102Groups.aActivateButton[45] = FALSE, input disabled if: DALI_Commissioning.fbPart102Groups.aActivateButton[45] = FALSE
            OnMouseClick: execute { DALI_Commissioning.fbPart102Groups.aButtonClick[45] := TRUE; }
        Textfield (405,255 50x30), "46", colour toggle: DALI_Commissioning.fbPart102Groups.aShowAlarmState[46] = TRUE, invisible if: DALI_Commissioning.fbPart102Groups.aActivateButton[46] = FALSE, input disabled if: DALI_Commissioning.fbPart102Groups.aActivateButton[46] = FALSE
            OnMouseClick: execute { DALI_Commissioning.fbPart102Groups.aButtonClick[46] := TRUE; }
        Textfield (470,255 50x30), "47", colour toggle: DALI_Commissioning.fbPart102Groups.aShowAlarmState[47] = TRUE, invisible if: DALI_Commissioning.fbPart102Groups.aActivateButton[47] = FALSE, input disabled if: DALI_Commissioning.fbPart102Groups.aActivateButton[47] = FALSE
            OnMouseClick: execute { DALI_Commissioning.fbPart102Groups.aButtonClick[47] := TRUE; }
        Textfield (15,300 50x30), "48", colour toggle: DALI_Commissioning.fbPart102Groups.aShowAlarmState[48] = TRUE, invisible if: DALI_Commissioning.fbPart102Groups.aActivateButton[48] = FALSE, input disabled if: DALI_Commissioning.fbPart102Groups.aActivateButton[48] = FALSE
            OnMouseClick: execute { DALI_Commissioning.fbPart102Groups.aButtonClick[48] := TRUE; }
        Textfield (80,300 50x30), "49", colour toggle: DALI_Commissioning.fbPart102Groups.aShowAlarmState[49] = TRUE, invisible if: DALI_Commissioning.fbPart102Groups.aActivateButton[49] = FALSE, input disabled if: DALI_Commissioning.fbPart102Groups.aActivateButton[49] = FALSE
            OnMouseClick: execute { DALI_Commissioning.fbPart102Groups.aButtonClick[49] := TRUE; }
        Textfield (145,300 50x30), "50", colour toggle: DALI_Commissioning.fbPart102Groups.aShowAlarmState[50] = TRUE, invisible if: DALI_Commissioning.fbPart102Groups.aActivateButton[50] = FALSE, input disabled if: DALI_Commissioning.fbPart102Groups.aActivateButton[50] = FALSE
            OnMouseClick: execute { DALI_Commissioning.fbPart102Groups.aButtonClick[50] := TRUE; }
        Textfield (210,300 50x30), "51", colour toggle: DALI_Commissioning.fbPart102Groups.aShowAlarmState[51] = TRUE, invisible if: DALI_Commissioning.fbPart102Groups.aActivateButton[51] = FALSE, input disabled if: DALI_Commissioning.fbPart102Groups.aActivateButton[51] = FALSE
            OnMouseClick: execute { DALI_Commissioning.fbPart102Groups.aButtonClick[51] := TRUE; }
        Textfield (275,300 50x30), "52", colour toggle: DALI_Commissioning.fbPart102Groups.aShowAlarmState[52] = TRUE, invisible if: DALI_Commissioning.fbPart102Groups.aActivateButton[52] = FALSE, input disabled if: DALI_Commissioning.fbPart102Groups.aActivateButton[52] = FALSE
            OnMouseClick: execute { DALI_Commissioning.fbPart102Groups.aButtonClick[52] := TRUE; }
        Textfield (340,300 50x30), "53", colour toggle: DALI_Commissioning.fbPart102Groups.aShowAlarmState[53] = TRUE, invisible if: DALI_Commissioning.fbPart102Groups.aActivateButton[53] = FALSE, input disabled if: DALI_Commissioning.fbPart102Groups.aActivateButton[53] = FALSE
            OnMouseClick: execute { DALI_Commissioning.fbPart102Groups.aButtonClick[53] := TRUE; }
        Textfield (405,300 50x30), "54", colour toggle: DALI_Commissioning.fbPart102Groups.aShowAlarmState[54] = TRUE, invisible if: DALI_Commissioning.fbPart102Groups.aActivateButton[54] = FALSE, input disabled if: DALI_Commissioning.fbPart102Groups.aActivateButton[54] = FALSE
            OnMouseClick: execute { DALI_Commissioning.fbPart102Groups.aButtonClick[54] := TRUE; }
        Textfield (470,300 50x30), "55", colour toggle: DALI_Commissioning.fbPart102Groups.aShowAlarmState[55] = TRUE, invisible if: DALI_Commissioning.fbPart102Groups.aActivateButton[55] = FALSE, input disabled if: DALI_Commissioning.fbPart102Groups.aActivateButton[55] = FALSE
            OnMouseClick: execute { DALI_Commissioning.fbPart102Groups.aButtonClick[55] := TRUE; }
        Textfield (15,345 50x30), "56", colour toggle: DALI_Commissioning.fbPart102Groups.aShowAlarmState[56] = TRUE, invisible if: DALI_Commissioning.fbPart102Groups.aActivateButton[56] = FALSE, input disabled if: DALI_Commissioning.fbPart102Groups.aActivateButton[56] = FALSE
            OnMouseClick: execute { DALI_Commissioning.fbPart102Groups.aButtonClick[56] := TRUE; }
        Textfield (80,345 50x30), "57", colour toggle: DALI_Commissioning.fbPart102Groups.aShowAlarmState[57] = TRUE, invisible if: DALI_Commissioning.fbPart102Groups.aActivateButton[57] = FALSE, input disabled if: DALI_Commissioning.fbPart102Groups.aActivateButton[57] = FALSE
            OnMouseClick: execute { DALI_Commissioning.fbPart102Groups.aButtonClick[56] := TRUE; }
        Textfield (145,345 50x30), "58", colour toggle: DALI_Commissioning.fbPart102Groups.aShowAlarmState[58] = TRUE, invisible if: DALI_Commissioning.fbPart102Groups.aActivateButton[58] = FALSE, input disabled if: DALI_Commissioning.fbPart102Groups.aActivateButton[58] = FALSE
            OnMouseClick: execute { DALI_Commissioning.fbPart102Groups.aButtonClick[58] := TRUE; }
        Textfield (210,345 50x30), "59", colour toggle: DALI_Commissioning.fbPart102Groups.aShowAlarmState[59] = TRUE, invisible if: DALI_Commissioning.fbPart102Groups.aActivateButton[59] = FALSE, input disabled if: DALI_Commissioning.fbPart102Groups.aActivateButton[59] = FALSE
            OnMouseClick: execute { DALI_Commissioning.fbPart102Groups.aButtonClick[59] := TRUE; }
        Textfield (275,345 50x30), "60", colour toggle: DALI_Commissioning.fbPart102Groups.aShowAlarmState[60] = TRUE, invisible if: DALI_Commissioning.fbPart102Groups.aActivateButton[60] = FALSE, input disabled if: DALI_Commissioning.fbPart102Groups.aActivateButton[60] = FALSE
            OnMouseClick: execute { DALI_Commissioning.fbPart102Groups.aButtonClick[60] := TRUE; }
        Textfield (340,345 50x30), "61", colour toggle: DALI_Commissioning.fbPart102Groups.aShowAlarmState[61] = TRUE, invisible if: DALI_Commissioning.fbPart102Groups.aActivateButton[61] = FALSE, input disabled if: DALI_Commissioning.fbPart102Groups.aActivateButton[61] = FALSE
            OnMouseClick: execute { DALI_Commissioning.fbPart102Groups.aButtonClick[61] := TRUE; }
        Textfield (405,345 50x30), "62", colour toggle: DALI_Commissioning.fbPart102Groups.aShowAlarmState[62] = TRUE, invisible if: DALI_Commissioning.fbPart102Groups.aActivateButton[62] = FALSE, input disabled if: DALI_Commissioning.fbPart102Groups.aActivateButton[62] = FALSE
            OnMouseClick: execute { DALI_Commissioning.fbPart102Groups.aButtonClick[62] := TRUE; }
        Textfield (470,345 50x30), "63", colour toggle: DALI_Commissioning.fbPart102Groups.aShowAlarmState[63] = TRUE, invisible if: DALI_Commissioning.fbPart102Groups.aActivateButton[63] = FALSE, input disabled if: DALI_Commissioning.fbPart102Groups.aActivateButton[63] = FALSE
            OnMouseClick: execute { DALI_Commissioning.fbPart102Groups.aButtonClick[63] := TRUE; }
        WaitingSymbolFlower (230,170 70x70), invisible if: DALI_Commissioning.fbPart102Groups.bHideWaitSymbol
    Button (610,400 150x40), "Read"
        OnMouseClick: execute { DALI_Commissioning.fbPart102Groups.bRead := TRUE; }
    Button (610,450 150x40), "Write"
        OnMouseClick: execute { DALI_Commissioning.fbPart102Groups.bWrite := TRUE; }
    Button (610,100 150x40), "Switch On"
        OnMouseClick: execute { DALI_Commissioning.fbPart102Groups.bSwitchOn := TRUE; }
    Button (610,150 150x40), "Switch Off"
        OnMouseClick: execute { DALI_Commissioning.fbPart102Groups.bSwitchOff := TRUE; }
    Group (320,5 210x40)
        Textfield (0,0 120x40), "Choose group:"
        Button (130,0 80x40), "%s", text variable: DALI_Commissioning.fbPart102Groups.nGroupAddress
            OnMouseClick: write the text variable via Default, min 0, max 15, title "Choose group"
    Group (10,5 170x40)
        Textfield (0,0 110x40), "DALI Line:"
        Button (90,0 80x40), "%d", text variable: GVL_Internal.nDALILine
            OnMouseClick: write the text variable via Default, min 1, max 10, title "Choose line"
END_VISUALIZATION

// ---- POUs/DALI/DALI_Setup/VISUs/Visu_DALICommissioning/Visu_Part102MemoryBank.TcVIS
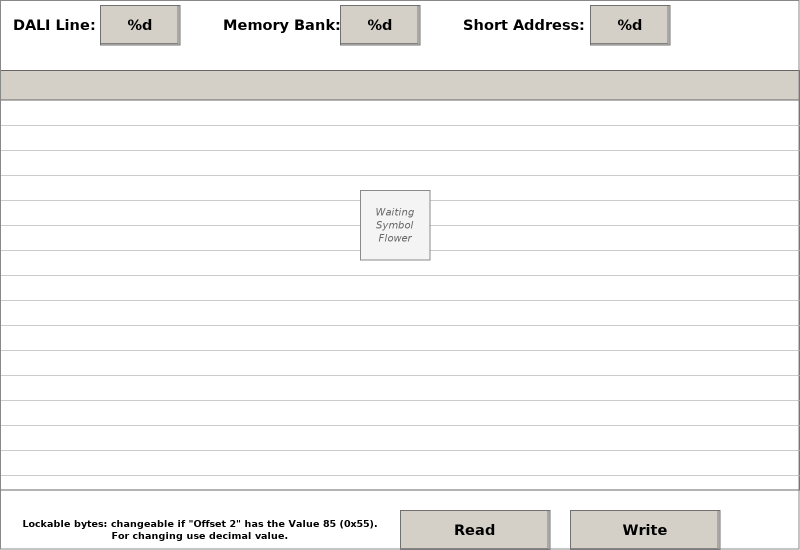
VISUALIZATION Visu_Part102MemoryBank  // 800x550
    Table (0,70 800x420), data array: DALI_Commissioning.fbPart102MemoryPages.aMemoryBank
        p1137915858: DALI_Commissioning.fbPart102MemoryPages.nOffset
        p3854506369: DALI_Commissioning.fbPart102MemoryPages.aMemoryBank[INDEX].sOffset
        p1892666644: DALI_Commissioning.fbPart102MemoryPages.aMemoryBank[INDEX].sName
        p338671338: DALI_Commissioning.fbPart102MemoryPages.aMemoryBank[INDEX].nValueDec
        p2170511999: DALI_Commissioning.fbPart102MemoryPages.aMemoryBank[INDEX].nValueHex
        p1755163831: Value Dec
        p4092479075: Value Hex
        Columns.Column.[0].Template: DALI_Commissioning.fbPart102MemoryPages.aNoValue[INDEX]
        Columns.Column.[1].Template: DALI_Commissioning.fbPart102MemoryPages.aNoValue[INDEX]
        Columns.Column.[2].Template: DALI_Commissioning.fbPart102MemoryPages.aNoValue[INDEX]; OnMouseClick: write the text variable via Default, min 0, max 255, title "Lockable variable decimal"
        Columns.Column.[3].Template: DALI_Commissioning.fbPart102MemoryPages.aNoValue[INDEX]; OnMouseClick: write the text variable via Default, title "Lockable variable hexadecimal"
    Button (400,510 150x40), "Read"
        OnMouseClick: execute { DALI_Commissioning.fbPart102MemoryPages.bRead := TRUE; }
    Button (570,510 150x40), "Write"
        OnMouseClick: execute { DALI_Commissioning.fbPart102MemoryPages.bWrite := TRUE; }
    Textfield (15,510 370x40), "Lockable bytes: changeable if "Offset 2" has the Value 85 (0x55). For changing use decimal value."
    WaitingSymbolFlower (360,190 70x70), invisible if: DALI_Commissioning.fbPart102MemoryPages.bHideWaitSymbol
    Textfield (460,5 130x40), "Short Address:"
    Button (590,5 80x40), "%d", text variable: DALI_Commissioning.fbPart102MemoryPages.nAddress
        OnMouseClick: write the text variable via Default, min 0, max 63, title "Insert Short Address"
    Textfield (220,5 120x40), "Memory Bank:"
    Button (340,5 80x40), "%d", text variable: DALI_Commissioning.fbPart102MemoryPages.nMemoryBank
        OnMouseClick: write the text variable via Default, min 0, max 255, title "Insert Memory Bank"
    Group (10,5 170x40)
        Textfield (0,0 110x40), "DALI Line:"
        Button (90,0 80x40), "%d", text variable: GVL_Internal.nDALILine
            OnMouseClick: write the text variable via Default, min 1, max 10, title "Choose line"
END_VISUALIZATION

// ---- POUs/DALI/DALI_Setup/VISUs/Visu_DALICommissioning/Visu_Part102Parameters.TcVIS
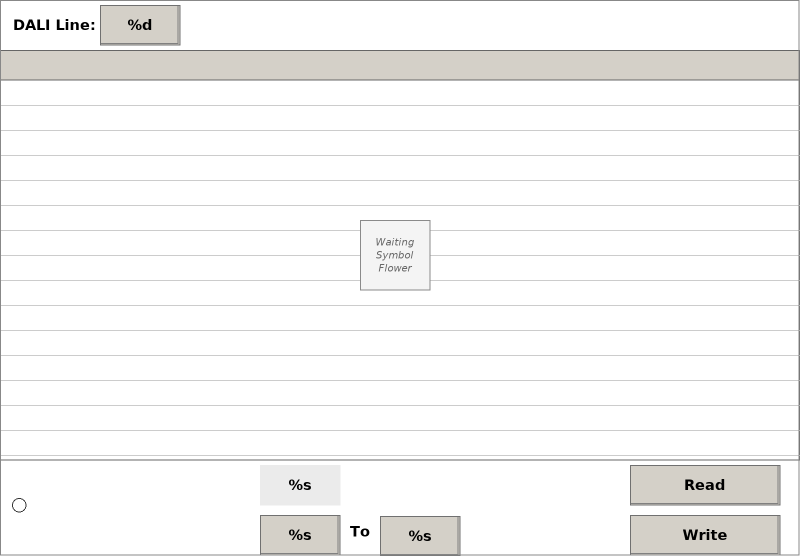
VISUALIZATION Visu_Part102Parameters  // 800x556
    Table (0,50 800x410), data array: DALI_Commissioning.fbPart102Parameters.aParameters
        p1137915858: DALI_Commissioning.fbPart102Parameters.nSelectedAddress
        p3854506369: DALI_Commissioning.fbPart102Parameters.aParameters[INDEX].nShortAddress
        p1892666644: DALI_Commissioning.fbPart102Parameters.aParameters[INDEX].nActualLevel
        p338671338: DALI_Commissioning.fbPart102Parameters.aParameters[INDEX].nMinLevel
        p2170511999: DALI_Commissioning.fbPart102Parameters.aParameters[INDEX].nMaxLevel
        p3723444502: DALI_Commissioning.fbPart102Parameters.aParameters[INDEX].eFadeRate
        p1218418051: DALI_Commissioning.fbPart102Parameters.aParameters[INDEX].eFadeTime
        p746581629: DALI_Commissioning.fbPart102Parameters.aParameters[INDEX].nPowerOnLevel
        p3104783080: DALI_Commissioning.fbPart102Parameters.aParameters[INDEX].nSystemFailureLevel
        p2501879983: DALI_Commissioning.fbPart102Parameters.aParameters[INDEX].nPhysicalMinimum
        p7306298: DALI_Commissioning.fbPart102Parameters.aParameters[INDEX].sDeviceTypes
        Columns.Column.[1].Template: OnMouseClick: write the text variable via Default, min 0, max 254, title "MinLevel"
        Columns.Column.[2].Template: OnMouseClick: write the text variable via Default, min 1, max 254, title "MaxLevel"
        Columns.Column.[3].Template: OnMouseClick: write the text variable via Default, min 0, max 254, title "FadeRate"
        Columns.Column.[4].Template: OnMouseClick: write the text variable via Default, min 1, max 15, title "Fade Rate"
        Columns.Column.[5].Template: OnMouseClick: write the text variable via Default, min 0, max 15, title "Fade Time"
        Columns.Column.[6].Template: OnMouseClick: write the text variable via Default, min 1, max 254, title "Power On Level"
        Columns.Column.[7].Template: OnMouseClick: write the text variable via Default, min 0, max 255, title "System Failure Level"
    RadioButton (10,455 254x100), variable: DALI_Commissioning.fbPart102Parameters.nAddressRange
        Areas[0]: Text=Single Short Address
        Areas[1]: Text=Short Address Range
    Textfield (335,516 50x31), "To"
    Button (630,465 150x40), "Read"
        OnMouseClick: execute { DALI_Commissioning.fbPart102Parameters.bRead := TRUE; }
    Button (630,515 150x40), "Write"
        OnMouseClick: execute { DALI_Commissioning.fbPart102Parameters.bWrite := TRUE; }
    Button (260,515 80x40), "%s", text variable: DALI_Commissioning.fbPart102Parameters.nStartAddress
        OnMouseClick: write the text variable via Default, min 0, max 63, title "Insert Short Address"
    Button (380,516 80x40), "%s", text variable: DALI_Commissioning.fbPart102Parameters.nEndAddress
        OnMouseClick: write the text variable via Default, min 0, max 63, title "Insert Short Address"
    Textfield (260,465 80x40), "%s", tooltip "Please select the desired Short Address in the table above.", text variable: DALI_Commissioning.fbPart102Parameters.nSelectedAddress
    WaitingSymbolFlower (360,220 70x70), invisible if: DALI_Commissioning.fbPart102Parameters.bHideWaitSymbol
    Group (10,5 170x40)
        Textfield (0,0 110x40), "DALI Line:"
        Button (90,0 80x40), "%d", text variable: GVL_Internal.nDALILine
            OnMouseClick: write the text variable via Default, min 1, max 10, title "Choose line"
END_VISUALIZATION

// ---- POUs/DALI/DALI_Setup/VISUs/Visu_DALICommissioning/Visu_Part102SetFading.TcVIS
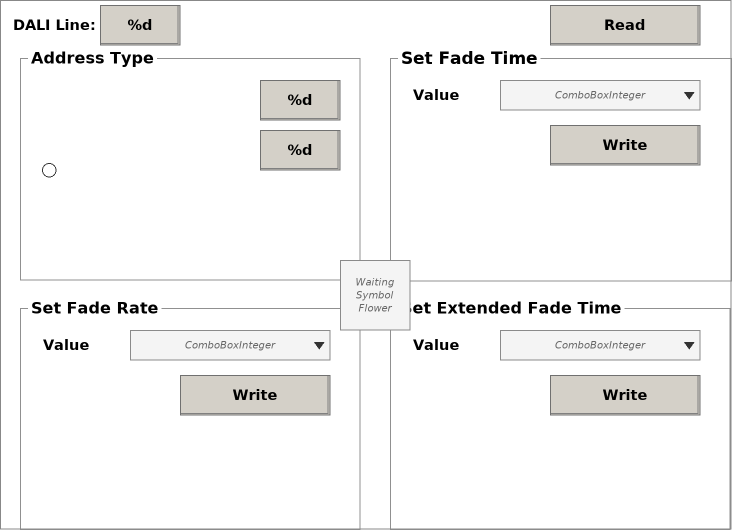
VISUALIZATION Visu_Part102SetFading  // 732x530
    GroupBox (390,50 342x231), "Set Fade Time"
        Textfield (20,30 100x30), "Value"
        ComboBoxInteger (110,30 200x30), variable: DALI_Commissioning.fbPart102SetFading.eFadeTime, text list: 'FadeTime'
        Button (160,75 150x40), "Write"
            OnMouseClick: execute { DALI_Commissioning.fbPart102SetFading.bWriteFadeTime := TRUE; }
    GroupBox (20,50 340x230), "Address Type"
        Button (240,30 80x40), "%d", text variable: DALI_Commissioning.fbPart102SetFading.nShortAddress
            OnMouseClick: write the text variable via Default, min 0, max 63, title "Insert Short Address"
        RadioButton (20,20 190x200), variable: DALI_Commissioning.fbPart102SetFading.eAddressType
            Areas[0]: Text=Short Address
            Areas[1]: Text=Group Address
            Areas[2]: Text=Broadcast
            Areas[3]: Text=Unaddressed
        Button (240,80 80x40), "%d", text variable: DALI_Commissioning.fbPart102SetFading.nGroupAddress
            OnMouseClick: write the text variable via Default, min 0, max 15, title "Insert Group Address"
    GroupBox (20,300 340x230), "Set Fade Rate"
        Textfield (20,30 100x30), "Value"
        ComboBoxInteger (110,30 200x30), variable: DALI_Commissioning.fbPart102SetFading.eFadeRate, text list: 'FadeRate'
        Button (160,75 150x40), "Write"
            OnMouseClick: execute { DALI_Commissioning.fbPart102setFading.bWriteFadeRate := TRUE; }
    GroupBox (390,300 340x230), "Set Extended Fade Time"
        Textfield (20,30 100x30), "Value"
        ComboBoxInteger (110,30 200x30), tooltip "Extended Fade Time only valid if Fade Time equals 0!", variable: DALI_Commissioning.fbPart102SetFading.eExtendedFadeTime, input disabled if: DALI_Commissioning.fbPart102SetFading.bNoFadeTime, text list: 'ExtendedFadeTime'
        Button (160,75 150x40), "Write", tooltip "Extended Fade Time only valid if Fade Time equals 0!", invisible if: DALI_Commissioning.fbPart102SetFading.bNoFadeTime, input disabled if: DALI_Commissioning.fbPart102SetFading.bNoFadeTime
            OnMouseClick: execute { DALI_Commissioning.fbPart102SetFading.bWriteExtendedFadeTime:=true; }
    Button (550,5 150x40), "Read", tooltip "Reads all Fading Parameters", invisible if: ( DALI_Commissioning.fbPart102SetFading.eAddressType >=1), input disabled if: ( DALI_Commissioning.fbPart102SetFading.eAddressType >=1)
        OnMouseClick: execute { DALI_Commissioning.fbPart102SetFading.bRead := TRUE; }
    WaitingSymbolFlower (340,260 70x70), invisible if: DALI_Commissioning.fbPart102SetFading.bHideWaitSymbol
    Group (10,5 170x40)
        Textfield (0,0 110x40), "DALI Line:"
        Button (90,0 80x40), "%d", text variable: GVL_Internal.nDALILine
            OnMouseClick: write the text variable via Default, min 1, max 10, title "Choose line"
END_VISUALIZATION

// ---- POUs/DALI/DALI_Setup/VISUs/Visu_DALICommissioning/Visu_Part103Addressing.TcVIS
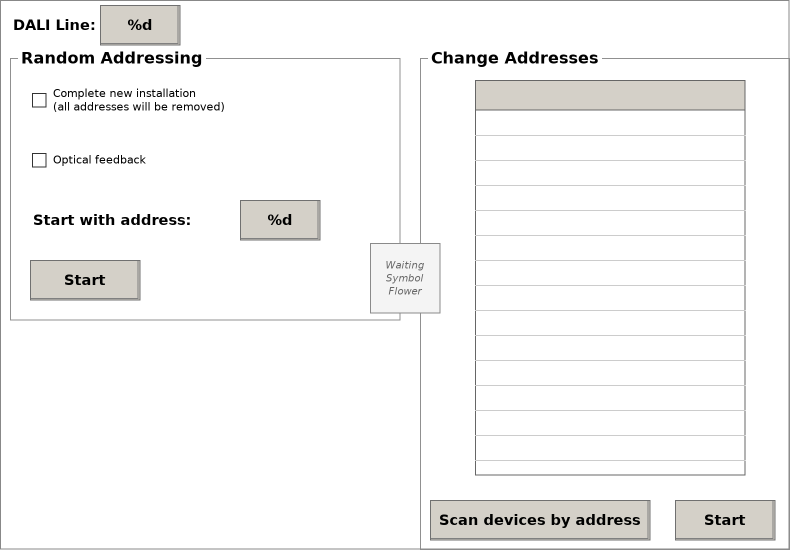
VISUALIZATION Visu_Part103Addressing  // 790x550
    GroupBox (420,50 370x500), "Change Addresses"
        Table (55,30 270x395), data array: DALI_Commissioning.fbPart103Addressing.aChangeAddressList
            p3854506369: DALI_Commissioning.fbPart103Addressing.aChangeAddressList[INDEX].nOldAddress
            p1892666644: DALI_Commissioning.fbPart103Addressing.aChangeAddressList[INDEX].nNewAddress
            p338671338: DALI_Commissioning.fbPart103Addressing.aChangeAddressList[INDEX].nRandomAddress
            p2170511999: DALI_Commissioning.fbPart103Addressing.aChangeAddressList[INDEX].nErrors
            Columns.Column.[0].Template: DALI_Commissioning.fbPart103Addressing.aNoShortAddress[INDEX]
            Columns.Column.[1].Template: DALI_Commissioning.fbPart103Addressing.aNoShortAddress[INDEX]; OnMouseClick: write the text variable via Default, min 0, max 63, title "New Short Address"
        Button (255,450 100x40), "Start"
            OnMouseClick: execute { DALI_Commissioning.fbPart103Addressing.bStartChangeAddress := TRUE; }
        Button (10,450 220x40), "Scan devices by address"
            OnMouseClick: execute { DALI_Commissioning.fbPart103Addressing.bScanDevices := TRUE; }
    GroupBox (10,50 390x270), "Random Addressing"
        Button (20,210 110x40), "Start"
            OnMouseClick: execute { DALI_Commissioning.fbPart103Addressing.bStartRandomAddressing := TRUE; }
        Checkbox (20,30 360x40), "Complete new installation (all addresses will be removed)", variable: DALI_Commissioning.fbPart103Addressing.bNewInstallation
        Checkbox (20,90 360x40), "Optical feedback", variable: DALI_Commissioning.fbPart103Addressing.bOpticalFeedback
        Textfield (20,150 200x40), "Start with address:"
        Button (230,150 80x40), "%d", text variable: DALI_Commissioning.fbPart103Addressing.nStartAddress
            OnMouseClick: write DALI_Commissioning.fbPart103Addressing.nStartAddress via Default, min 0, max 63, title "Insert Short Address"
    WaitingSymbolFlower (370,243 70x70), invisible if: DALI_Commissioning.fbPart103Addressing.bHideWaitSymbol
    Group (10,5 170x40)
        Textfield (0,0 110x40), "DALI Line:"
        Button (90,0 80x40), "%d", text variable: GVL_Internal.nDALILine
            OnMouseClick: write the text variable via Default, min 1, max 10, title "Choose line"
END_VISUALIZATION

// ---- POUs/DALI/DALI_Setup/VISUs/Visu_DALICommissioning/Visu_Part103Identify.TcVIS
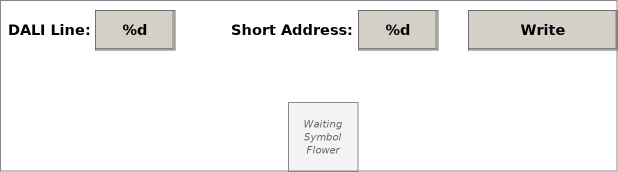
VISUALIZATION Visu_Part103Identify  // 618x172
    Button (468,10 150x40), "Write"
        OnMouseClick: execute { DALI_Commissioning.fbPart103IdentifyDevice.bWrite := TRUE; }
    WaitingSymbolFlower (288,102 70x70), invisible if: DALI_Commissioning.fbPart103MemoryPages.bHideWaitSymbol
    Textfield (228,10 130x40), "Short Address:"
    Button (358,10 80x40), "%d", text variable: DALI_Commissioning.fbPart103IdentifyDevice.nAddress
        OnMouseClick: write the text variable via Default, min 0, max 63, title "Insert Short Address"
    Group (5,10 170x40)
        Textfield (0,0 110x40), "DALI Line:"
        Button (90,0 80x40), "%d", text variable: GVL_Internal.nDALILine
            OnMouseClick: write the text variable via Default, min 1, max 10, title "Choose line"
END_VISUALIZATION

// ---- POUs/DALI/DALI_Setup/VISUs/Visu_DALICommissioning/Visu_Part103Parameters.TcVIS
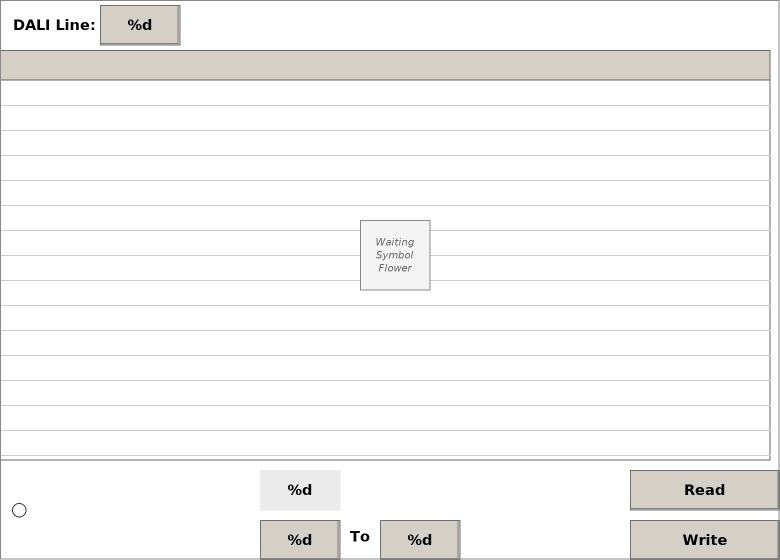
VISUALIZATION Visu_Part103Parameters  // 780x560
    Table (0,50 770x410), data array: DALI_Commissioning.fbPart103Parameters.aParameters
        p1137915858: DALI_Commissioning.fbPart103Parameters.nSelectedAddress
        p3854506369: DALI_Commissioning.fbPart103Parameters.aParameters[INDEX].nOperatingMode
        p1892666644: DALI_Commissioning.fbPart103Parameters.aParameters[INDEX].sInstanceType0
        p338671338: DALI_Commissioning.fbPart103Parameters.aParameters[INDEX].sInstanceType1
        p2170511999: DALI_Commissioning.fbPart103Parameters.aParameters[INDEX].sInstanceType2
        p3723444502: DALI_Commissioning.fbPart103Parameters.aParameters[INDEX].sInstanceType3
        p1218418051: DALI_Commissioning.fbPart103Parameters.aParameters[INDEX].sInstanceType4
        p511219082: IT0 (Generic Input)
        p1755163831: IT1 (PushButton)
        p4092479075: IT2 (Absolute Input)
        p2237128397: IT3 (Occupancy)
        p505689113: IT4 (Light Sensor)
        Columns.Column.[0].Template: OnMouseClick: write the text variable via Default, min 0, max 255, title "Insert Operating Mode 0, 128-255"
    RadioButton (10,460 230x100), variable: DALI_Commissioning.fbPart103Parameters.nAddressRange
        Areas[0]: Text=Single Short Address
        Areas[1]: Text=Short Address Range
    Textfield (260,470 80x40), "%d", text variable: DALI_Commissioning.fbPart103Parameters.nSelectedAddress
    Button (260,520 80x40), "%d", text variable: DALI_Commissioning.fbPart103Parameters.nStartAddress
        OnMouseClick: write the text variable via Default, min 0, max 63, title "Insert Short Address"
    Button (380,520 80x40), "%d", text variable: DALI_Commissioning.fbPart103Parameters.nEndAddress
        OnMouseClick: write the text variable via Default, min 0, max 63, title "Insert Short Address"
    Button (630,470 150x40), "Read"
        OnMouseClick: execute { DALI_Commissioning.fbPart103Parameters.bRead := true; }
    Button (630,520 150x40), "Write"
        OnMouseClick: execute { DALI_Commissioning.fbPart103Parameters.bWrite := true; }
    Textfield (335,521 50x31), "To"
    WaitingSymbolFlower (360,220 70x70), invisible if: DALI_Commissioning.fbPart103Parameters.bHideWaitSymbol
    Group (10,5 170x40)
        Textfield (0,0 110x40), "DALI Line:"
        Button (90,0 80x40), "%d", text variable: GVL_Internal.nDALILine
            OnMouseClick: write the text variable via Default, min 1, max 10, title "Choose line"
END_VISUALIZATION

// ---- POUs/DALI/DALI_Setup/VISUs/Visu_DALICommissioning/Visu_Part202.TcVIS
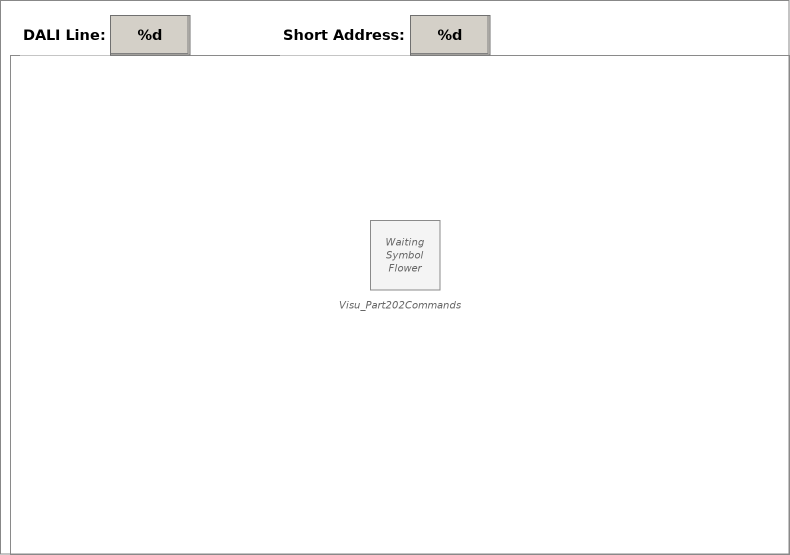
VISUALIZATION Visu_Part202  // 790x555
    TabControl (10,55 780x500)
        shows Visu_Part202Commands()
        shows Visu_Part202Status()
        shows Visu_Part202Parameters()
        [0]: TabTitle=Commands
        [1]: TabTitle=Status
        [2]: TabTitle=Parameters
    Group (280,15 210x40)
        Textfield (0,0 130x40), "Short Address:"
        Button (130,0 80x40), "%d", text variable: DALI_Commissioning.fbPart202Emergency.nAddress
            OnMouseClick: write the text variable via Default, min 0, max 63, title "Insert Short Address"
    Group (20,15 170x40)
        Textfield (0,0 110x40), "DALI Line:"
        Button (90,0 80x40), "%d", text variable: GVL_Internal.nDALILine
            OnMouseClick: write the text variable via Default, min 1, max 10, title "Choose line"
    WaitingSymbolFlower (370,220 70x70), invisible if: DALI_Commissioning.fbPart202Emergency.bHideWaitSymbol
END_VISUALIZATION

// ---- POUs/DALI/DALI_Setup/VISUs/Visu_DALICommissioning/Visu_Part202Parameters.TcVIS
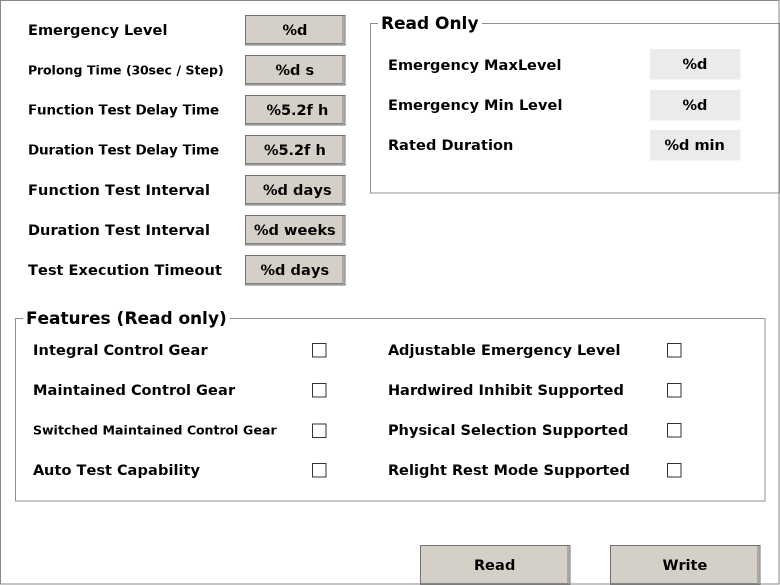
VISUALIZATION Visu_Part202Parameters  // 780x585
    Button (610,545 150x40), "Write"
        OnMouseClick: execute { DALI_Commissioning.fbPart202Emergency.bWrite:=TRUE; }
    GroupBox (15,310 750x191), "Features (Read only)"
        Textfield (15,25 250x30), "Integral Control Gear"
        Textfield (15,65 250x30), "Maintained Control Gear"
        Checkbox (295,105 30x31), variable: DALI_Commissioning.fbPart202Emergency.bSwitchtedMaintainedControlGear, input disabled if: TRUE
        Checkbox (295,25 30x30), variable: DALI_Commissioning.fbPart202Emergency.bIntegralControlGear, input disabled if: TRUE
        Checkbox (295,65 30x30), variable: DALI_Commissioning.fbPart202Emergency.bMaintainedControlGear, input disabled if: TRUE
        Textfield (370,105 250x30), "Physical Selection Supported"
        Textfield (15,145 250x30), "Auto Test Capability"
        Textfield (370,25 250x30), "Adjustable Emergency Level"
        Textfield (370,65 250x30), "Hardwired Inhibit Supported"
        Textfield (370,145 250x30), "Relight Rest Mode Supported"
        Checkbox (650,25 30x30), variable: DALI_Commissioning.fbPart202Emergency.bAdjustableEmergencyLevel, input disabled if: TRUE
        Checkbox (650,65 30x30), variable: DALI_Commissioning.fbPart202Emergency.bHardwiredInhibitSupported, input disabled if: TRUE
        Checkbox (650,105 30x30), variable: DALI_Commissioning.fbPart202Emergency.bPhysicalSelectionSupported, input disabled if: TRUE
        Checkbox (650,145 30x30), variable: DALI_Commissioning.fbPart202Emergency.bRelightinRestModeSupported, input disabled if: TRUE
        Textfield (15,105 250x30), "Switched Maintained Control Gear"
        Checkbox (295,145 30x30), variable: DALI_Commissioning.fbPart202Emergency.bAutoTestCapability, input disabled if: TRUE
    Textfield (25,15 200x30), "Emergency Level"
    Textfield (25,95 200x30), "Function Test Delay Time"
    Textfield (25,135 200x30), "Duration Test Delay Time"
    Button (245,15 100x30), "%d", text variable: DALI_Commissioning.fbPart202Emergency.nEmergencyLevel
        OnMouseClick: write the text variable via Default, min 0, max 255, title "Emergency Level"
    Button (245,95 100x30), "%5.2f h", text variable: DALI_Commissioning.fbPart205Incandescent.fLoadRating
        OnMouseClick: write the text variable via Default, min 0, max 16384, title "Function Test Delay Time"
    Button (245,135 100x30), "%5.2f h", text variable: DALI_Commissioning.fbPart202Emergency.fDurationTestDelayTimeVisu
        OnMouseClick: write the text variable via Default, min 0, max 16384, title "Duration Test Delay Time"
    Textfield (25,55 200x30), "Prolong Time (30sec / Step)"
    Button (245,55 100x30), "%d s", text variable: DALI_Commissioning.fbPart202Emergency.nProlongTime
        OnMouseClick: write the text variable via Default, min 0, max 255, title "Prolong Time"
    Textfield (25,255 200x30), "Test Execution Timeout"
    Button (245,255 100x30), "%d days", text variable: DALI_Commissioning.fbPart202Emergency.nTestExecutionTimeout
        OnMouseClick: write the text variable via Default, min 0, max 255, title "Test Execution Timeout"
    GroupBox (370,15 410x178), "Read Only"
        Textfield (15,115 220x30), "Rated Duration"
        Textfield (15,75 220x30), "Emergency Min Level"
        Textfield (15,35 220x30), "Emergency MaxLevel"
        Textfield (280,34 90x30), "%d", text variable: DALI_Commissioning.fbPart202Emergency.nEmergencyMaxLevel
        Textfield (280,75 90x30), "%d", text variable: DALI_Commissioning.fbPart202Emergency.nEmergencyMinLevel
        Textfield (280,115 90x30), "%d min", text variable: DALI_Commissioning.fbPart202Emergency.nRatedDuration
    Textfield (25,175 200x30), "Function Test Interval"
    Textfield (25,215 200x30), "Duration Test Interval"
    Button (245,175 100x30), "%d days", text variable: DALI_Commissioning.fbPart202Emergency.nFunctionTestInterval
        OnMouseClick: write the text variable via Default, min 0, max 255, title "Function Test Delay Time"
    Button (245,215 100x30), "%d weeks", text variable: DALI_Commissioning.fbPart202Emergency.nDurationTestInterval
        OnMouseClick: write the text variable via Default, min 0, max 255, title "Duration Test Delay Time"
    Button (420,545 150x40), "Read"
        OnMouseClick: execute { DALI_Commissioning.fbPart202Emergency.bReadParameter:=TRUE; }
END_VISUALIZATION

// ---- POUs/DALI/DALI_Setup/VISUs/Visu_DALICommissioning/Visu_Part202Status.TcVIS
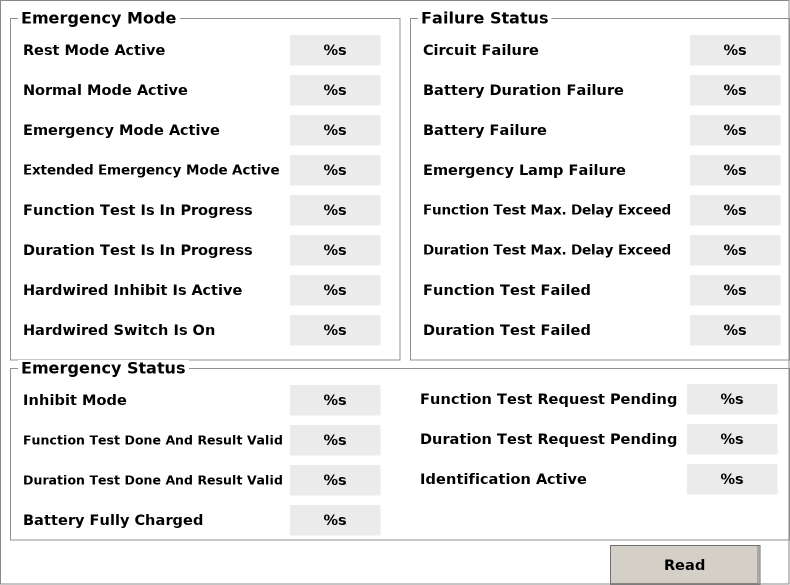
VISUALIZATION Visu_Part202Status  // 790x585
    Button (610,545 150x40), "Read"
        OnMouseClick: execute { DALI_Commissioning.fbPart202Emergency.bReadState:=TRUE; }
    GroupBox (10,10 390x350), "Emergency Mode"
        Textfield (10,145 260x30), "Extended Emergency Mode Active"
        Textfield (280,185 90x30), "%s", text variable: DALI_Commissioning.fbPart202Emergency.sFunctionTest
        Textfield (280,145 90x30), "%s", text variable: DALI_Commissioning.fbPart202Emergency.sExtendedEmergency
        Textfield (280,105 90x30), "%s", text variable: DALI_Commissioning.fbPart202Emergency.sEmergencyMode
        Textfield (280,65 90x30), "%s", text variable: DALI_Commissioning.fbPart202Emergency.sNormalMode
        Textfield (280,25 90x30), "%s", text variable: DALI_Commissioning.fbPart202Emergency.sRestMode
        Textfield (10,25 260x30), "Rest Mode Active"
        Textfield (10,65 260x30), "Normal Mode Active"
        Textfield (10,105 260x30), "Emergency Mode Active"
        Textfield (10,185 260x30), "Function Test Is In Progress"
        Textfield (10,225 260x30), "Duration Test Is In Progress"
        Textfield (10,265 260x30), "Hardwired Inhibit Is Active"
        Textfield (10,305 260x30), "Hardwired Switch Is On"
        Textfield (280,265 90x30), "%s", text variable: DALI_Commissioning.fbPart202Emergency.sHardwiredInhibit
        Textfield (280,305 90x30), "%s", text variable: DALI_Commissioning.fbPart202Emergency.sHardwiredSwitch
        Textfield (280,225 90x30), "%s", text variable: DALI_Commissioning.fbPart202Emergency.sDurationTest
    GroupBox (410,10 380x350), "Failure Status"
        Textfield (10,145 260x30), "Emergency Lamp Failure"
        Textfield (280,185 90x30), "%s", text variable: DALI_Commissioning.fbPart202Emergency.sFunctionTestExceed
        Textfield (280,145 90x30), "%s", text variable: DALI_Commissioning.fbPart202Emergency.sEmergencyLampFailure
        Textfield (280,105 90x30), "%s", text variable: DALI_Commissioning.fbPart202Emergency.sBatteryFailure
        Textfield (280,65 90x30), "%s", text variable: DALI_Commissioning.fbPart202Emergency.sBatteryDurationFailure
        Textfield (280,25 90x30), "%s", text variable: DALI_Commissioning.fbPart202Emergency.sCircuitFailure
        Textfield (10,25 260x30), "Circuit Failure"
        Textfield (10,65 260x30), "Battery Duration Failure"
        Textfield (10,105 260x30), "Battery Failure"
        Textfield (10,185 260x30), "Function Test Max. Delay Exceed"
        Textfield (10,225 260x30), "Duration Test Max. Delay Exceed"
        Textfield (10,265 260x30), "Function Test Failed"
        Textfield (10,305 260x30), "Duration Test Failed"
        Textfield (280,265 90x30), "%s", text variable: DALI_Commissioning.fbPart202Emergency.sFunctionTestFailed
        Textfield (280,305 90x30), "%s", text variable: DALI_Commissioning.fbPart202Emergency.sDurationTestFailed
        Textfield (280,225 90x30), "%s", text variable: DALI_Commissioning.fbPart202Emergency.sDurationTestExceed
    GroupBox (10,360 780x180), "Emergency Status"
        Textfield (10,145 260x30), "Battery Fully Charged"
        Textfield (677,24 90x30), "%s", text variable: DALI_Commissioning.fbPart202Emergency.sFunctionTestRequestPending
        Textfield (10,25 260x30), "Inhibit Mode"
        Textfield (10,65 260x30), "Function Test Done And Result Valid"
        Textfield (407,24 260x30), "Function Test Request Pending"
        Textfield (407,64 260x30), "Duration Test Request Pending"
        Textfield (407,104 260x30), "Identification Active"
        Textfield (677,104 90x30), "%s", text variable: DALI_Commissioning.fbPart202Emergency.sIdentificationActive
        Textfield (677,64 90x30), "%s", text variable: DALI_Commissioning.fbPart202Emergency.sDurationTestRequestPending
        Textfield (280,25 90x30), "%s", text variable: DALI_Commissioning.fbPart202Emergency.sInhibitMode
        Textfield (280,65 90x30), "%s", text variable: DALI_Commissioning.fbPart202Emergency.sFunctionTestDoneValid
        Textfield (280,145 90x30), "%s", text variable: DALI_Commissioning.fbPart202Emergency.sBatteryFullCharged
        Textfield (10,105 260x30), "Duration Test Done And Result Valid"
        Textfield (280,105 90x30), "%s", text variable: DALI_Commissioning.fbPart202Emergency.sDurationTestDoneValid
END_VISUALIZATION

// ---- POUs/DALI/DALI_Setup/VISUs/Visu_DALICommissioning/Visu_Part205.TcVIS
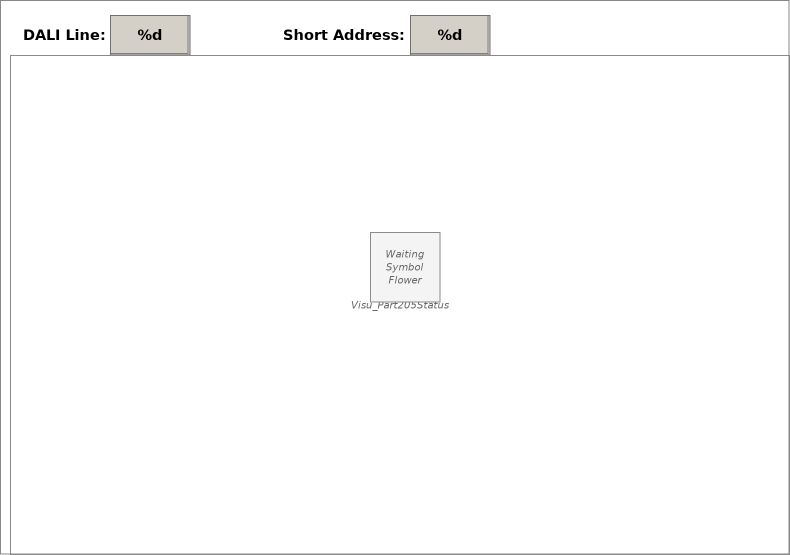
VISUALIZATION Visu_Part205  // 790x555
    Group (280,15 210x40)
        Textfield (0,0 130x40), "Short Address:"
        Button (130,0 80x40), "%d", text variable: DALI_Commissioning.fbPart205Incandescent.nAddress
            OnMouseClick: write the text variable via Default, min 0, max 63, title "Insert Short Address"
    Group (20,15 170x40)
        Textfield (0,0 110x40), "DALI Line:"
        Button (90,0 80x40), "%d", text variable: GVL_Internal.nDALILine
            OnMouseClick: write the text variable via Default, min 1, max 10, title "Choose line"
    TabControl (10,55 780x500)
        shows Visu_Part205Status()
        shows Visu_Part205Parameters()
        shows Visu_Part202Parameters()
        [0]: TabTitle=Status
        [1]: TabTitle=Parameters
        [2]: TabTitle=Parameters
    WaitingSymbolFlower (370,232 70x70), invisible if: DALI_Commissioning.fbPart205Incandescent.bHideWaitSymbol
END_VISUALIZATION

// ---- POUs/DALI/DALI_Setup/VISUs/Visu_DALICommissioning/Visu_Part205Status.TcVIS
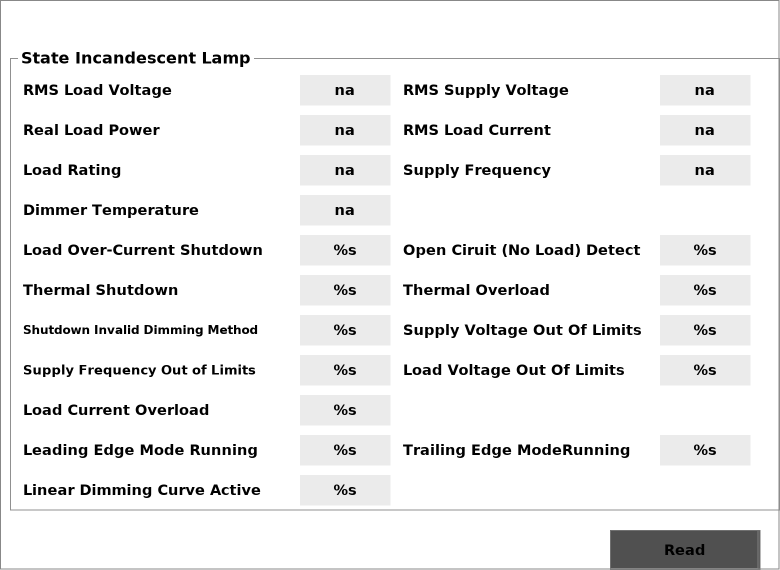
VISUALIZATION Visu_Part205Status  // 780x570
    Button (610,530 150x40), "Read"
        OnMouseClick: execute { DALI_Commissioning.fbPart205Incandescent.bReadStatus := TRUE; }
    GroupBox (10,50 770x460), "State Incandescent Lamp"
        Textfield (290,185 90x30), "%s", text variable: DALI_Commissioning.fbPart205Incandescent.sLoadOverCurrentShutdown
        Textfield (650,105 90x30), "%d Hz", text variable: DALI_Commissioning.fbPart205Incandescent.nSupplyFrequency
        Textfield (650,65 90x30), "%d %%", text variable: DALI_Commissioning.fbPart205Incandescent.nRMSLoadCurrent
        Textfield (650,25 90x30), "%d V", text variable: DALI_Commissioning.fbPart205Incandescent.nRMSSupplyVoltage
        Textfield (290,145 90x30), "%d °C", text variable: DALI_Commissioning.fbPart205Incandescent.nDimmerTemperature
        Textfield (290,105 90x30), "%2.1f mA", text variable: DALI_Commissioning.fbPart205Incandescent.fLoadRating
        Textfield (290,65 90x30), "%5.1f W", text variable: DALI_Commissioning.fbPart205Incandescent.fRealLoadPower
        Textfield (290,25 90x30), "%d V", text variable: DALI_Commissioning.fbPart205Incandescent.nRmsLoadVoltage
        Textfield (10,25 240x30), "RMS Load Voltage"
        Textfield (10,65 240x30), "Real Load Power", text variable: DALI_Commissioning.fbPart202Emergency.fFunctionTestDelayTimeVisu
        Textfield (10,145 240x30), "Dimmer Temperature"
        Textfield (10,105 240x30), "Load Rating"
        Textfield (10,185 240x30), "Load Over-Current Shutdown"
        Textfield (10,225 240x30), "Thermal Shutdown"
        Textfield (10,265 240x30), "Shutdown Invalid Dimming Method"
        Textfield (10,305 240x30), "Supply Frequency Out of Limits"
        Textfield (10,345 240x30), "Load Current Overload"
        Textfield (10,385 240x30), "Leading Edge Mode Running"
        Textfield (10,425 240x30), "Linear Dimming Curve Active"
        Textfield (290,265 90x30), "%s", text variable: DALI_Commissioning.fbPart205Incandescent.sInvalidDimmingMethod
        Textfield (290,305 90x30), "%s", text variable: DALI_Commissioning.fbPart205Incandescent.sSupplyFrequencyOutOfLimit
        Textfield (650,185 90x30), "%s", text variable: DALI_Commissioning.fbPart205Incandescent.sOpenCircuitDetection
        Textfield (650,225 90x30), "%s", text variable: DALI_Commissioning.fbPart205Incandescent.sThermalOverload
        Textfield (650,265 90x30), "%s", text variable: DALI_Commissioning.fbPart205Incandescent.sSupplyVoltageOutOfLimit
        Textfield (650,385 90x30), "%s", text variable: DALI_Commissioning.fbPart205Incandescent.sTrailingEdgeModeRunning
        Textfield (290,345 90x30), "%s", text variable: DALI_Commissioning.fbPart205Incandescent.sLoadCurrentOverload
        Textfield (290,385 90x30), "%s", text variable: DALI_Commissioning.fbPart205Incandescent.sLeadingEdgeModeRunning
        Textfield (290,425 90x30), "%s", text variable: DALI_Commissioning.fbPart205Incandescent.sLinearDimmingCurve
        Textfield (290,225 90x30), "%s", text variable: DALI_Commissioning.fbPart205Incandescent.sThermalShutdown
        Textfield (390,25 240x30), "RMS Supply Voltage"
        Textfield (390,65 240x30), "RMS Load Current"
        Textfield (390,105 240x30), "Supply Frequency"
        Textfield (390,185 240x30), "Open Ciruit (No Load) Detect"
        Textfield (390,225 240x30), "Thermal Overload"
        Textfield (390,265 240x30), "Supply Voltage Out Of Limits"
        Textfield (390,305 240x30), "Load Voltage Out Of Limits"
        Textfield (390,385 240x30), "Trailing Edge ModeRunning"
        Textfield (650,305 90x30), "%s", text variable: DALI_Commissioning.fbPart205Incandescent.sLoadVoltageOutOfLimit
        Textfield (290,25 90x30), "na", invisible if: not DALI_Commissioning.fbPart205Incandescent.bNoRmsLoadVoltage, input disabled if: true
        Textfield (290,65 90x30), "na", invisible if: not DALI_Commissioning.fbPart205Incandescent.bNoRealLoadPower, input disabled if: true
        Textfield (290,105 90x30), "na", invisible if: not DALI_Commissioning.fbPart205Incandescent.bNoLoadRating, input disabled if: true
        Textfield (290,145 90x30), "na", invisible if: not DALI_Commissioning.fbPart205Incandescent.bNoDimmerTemperature, input disabled if: true
        Textfield (650,25 90x30), "na", invisible if: not DALI_Commissioning.fbPart205Incandescent.bNoRMSSupplyVoltage, input disabled if: true
        Textfield (650,65 90x30), "na", invisible if: not DALI_Commissioning.fbPart205Incandescent.bNoRMSLoadCurrent, input disabled if: true
        Textfield (650,105 90x30), "na", invisible if: not DALI_Commissioning.fbPart205Incandescent.bNoSupplyFrequency, input disabled if: true
END_VISUALIZATION

// ---- POUs/DALI/DALI_Setup/VISUs/Visu_DALICommissioning/Visu_Part207.TcVIS
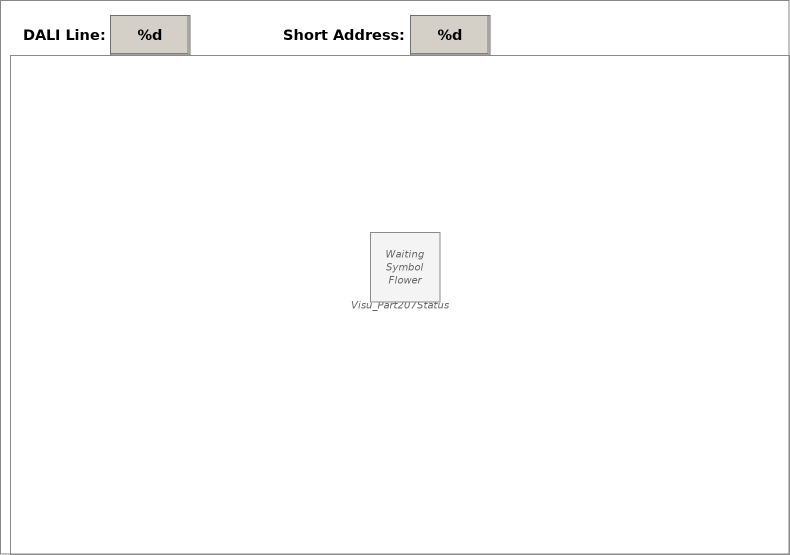
VISUALIZATION Visu_Part207  // 790x555
    Group (280,15 210x40)
        Textfield (0,0 130x40), "Short Address:"
        Button (130,0 80x40), "%d", text variable: DALI_Commissioning.fbPart207LED.nAddress
            OnMouseClick: write the text variable via Default, min 0, max 63, title "Insert Short Address"
    Group (20,15 170x40)
        Textfield (0,0 110x40), "DALI Line:"
        Button (90,0 80x40), "%d", text variable: GVL_Internal.nDALILine
            OnMouseClick: write the text variable via Default, min 1, max 10, title "Choose line"
    TabControl (10,55 780x500)
        shows Visu_Part207Status()
        shows Visu_Part207Parameters()
        shows Test()
        [0]: TabTitle=Status LED
        [1]: TabTitle=Parameters LED
        [2]: TabTitle=Paremeters LED
    WaitingSymbolFlower (370,232 70x70), invisible if: DALI_Commissioning.fbPart207LED.bHideWaitSymbol
END_VISUALIZATION

// ---- POUs/DALI/DALI_Setup/VISUs/Visu_DALICommissioning/Visu_Part207Parameters.TcVIS
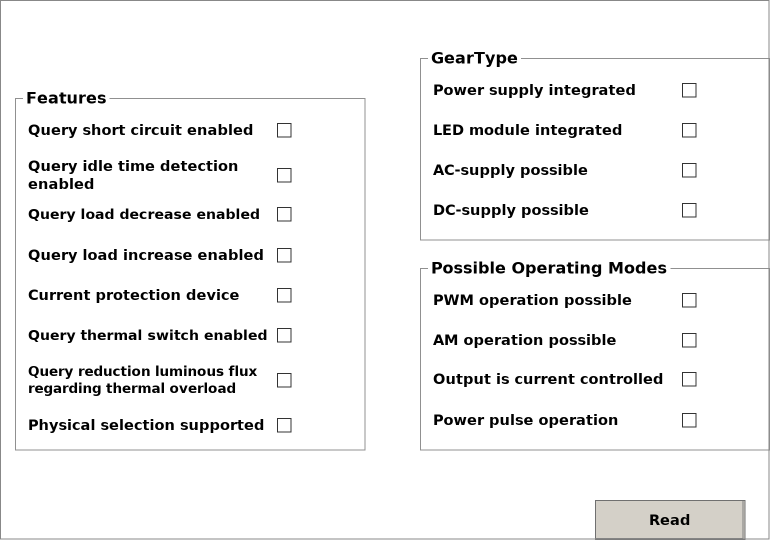
VISUALIZATION Visu_Part207Parameters  // 770x540
    Button (595,500 150x40), "Read"
        OnMouseClick: execute { DALI_Commissioning.fbPart207LED.bReadParameter:=TRUE; }
    GroupBox (420,50 350x190), "GearType"
        Textfield (10,25 220x30), "Power supply integrated"
        Checkbox (260,25 30x30), variable: DALI_Commissioning.fbPart207LED.bLEDPowerSupply, input disabled if: True
        Textfield (10,65 220x30), "LED module integrated"
        Textfield (10,145 220x30), "DC-supply possible"
        Textfield (10,105 220x30), "AC-supply possible"
        Checkbox (260,65 30x30), variable: DALI_Commissioning.fbPart207LED.bLEDModule, input disabled if: True
        Checkbox (260,145 30x30), variable: DALI_Commissioning.fbPart207LED.bDCSupply, input disabled if: True
        Checkbox (260,105 30x30), variable: DALI_Commissioning.fbPart207LED.bACSupply, input disabled if: True
    GroupBox (15,90 350x360), "Features"
        Textfield (10,25 240x30), "Query short circuit enabled"
        Checkbox (260,25 30x30), variable: DALI_Commissioning.fbPart207LED.bQueryShortCircuitEnabled, input disabled if: True
        Textfield (10,65 240x40), "Query idle time detection enabled"
        Textfield (10,150 240x30), "Query load increase enabled"
        Textfield (10,109 240x30), "Query load decrease enabled"
        Checkbox (260,70 30x30), variable: DALI_Commissioning.fbPart207LED.bQueryIdleTimeDetectionEnabled, input disabled if: True
        Checkbox (260,150 30x30), variable: DALI_Commissioning.fbPart207LED.bQueryLoadIncreaseEnabled, input disabled if: True
        Checkbox (260,109 30x30), variable: DALI_Commissioning.fbPart207LED.bQueryLoadDecreaseEnabled, input disabled if: True
        Textfield (10,190 240x30), "Current protection device"
        Checkbox (260,190 30x30), variable: DALI_Commissioning.fbPart207LED.bQueryCurrentProtectionDevicePresent, input disabled if: True
        Checkbox (260,230 30x30), variable: DALI_Commissioning.fbPart207LED.bQueryThermalSwitchEnabled, input disabled if: True
        Checkbox (260,275 30x30), variable: DALI_Commissioning.fbPart207LED.bQueryReductionOfLuminouFluxRegardingThermalOverloadEnabled, input disabled if: True
        Checkbox (260,320 30x30), variable: DALI_Commissioning.fbPart207LED.bPhysicalSelectionSupported, input disabled if: True
        Textfield (10,230 240x30), "Query thermal switch enabled"
        Textfield (10,270 240x40), "Query reduction luminous flux regarding thermal overload"
        Textfield (10,320 240x30), "Physical selection supported"
    GroupBox (420,260 350x190), "Possible Operating Modes", invisible if: DALI_Commissioning.fbPart207LED.bInvisible
        Checkbox (260,25 30x30), variable: DALI_Commissioning.fbPart207LED.bPWMOperation, input disabled if: True
        Textfield (10,65 240x30), "AM operation possible"
        Textfield (10,145 240x30), "Power pulse operation"
        Textfield (10,104 240x30), "Output is current controlled"
        Checkbox (260,65 30x30), variable: DALI_Commissioning.fbPart207LED.bAMOperation, input disabled if: True
        Checkbox (260,145 30x30), variable: DALI_Commissioning.fbPart207LED.bPowerPulseOperation, input disabled if: True
        Checkbox (260,104 30x30), variable: DALI_Commissioning.fbPart207LED.bOutputCurrentControlled, input disabled if: True
        Textfield (10,25 240x30), "PWM operation possible"
END_VISUALIZATION

// ---- POUs/DALI/DALI_Setup/VISUs/Visu_DALICommissioning/Visu_Part208Switching.TcVIS
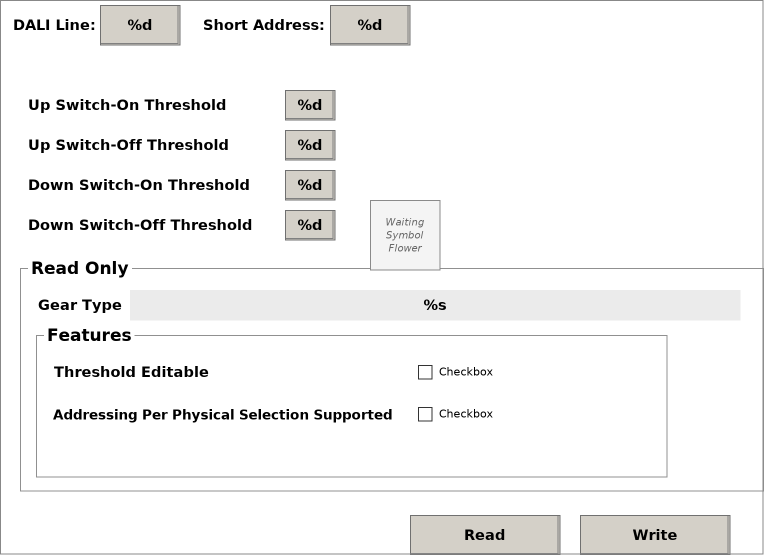
VISUALIZATION Visu_Part208Switching  // 764x555
    Group (200,5 210x40)
        Textfield (0,0 130x40), "Short Address:"
        Button (130,0 80x40), "%d", text variable: DALI_Commissioning.fbPart208Switching.nAddress
            OnMouseClick: write the text variable via Default, min 0, max 63, title "Insert Short Address"
    Group (10,5 170x40)
        Textfield (0,0 110x40), "DALI Line:"
        Button (90,0 80x40), "%d", text variable: GVL_Internal.nDALILine
            OnMouseClick: write the text variable via Default, min 1, max 10, title "Choose line"
    Textfield (25,90 250x30), "Up Switch-On Threshold"
    Textfield (25,130 250x30), "Up Switch-Off Threshold"
    Textfield (25,170 250x30), "Down Switch-On Threshold"
    Textfield (25,210 250x30), "Down Switch-Off Threshold"
    GroupBox (20,260 744x231), "Read Only"
        Textfield (15,30 250x30), "Gear Type"
        Textfield (110,30 610x30), "%s", text variable: DALI_Commissioning.fbPart208Switching.sGearType
        GroupBox (16,67 631x150), "Features"
            Checkbox (380,30 30x30), "Checkbox", variable: DALI_Commissioning.fbPart208Switching.bThreshold, input disabled if: TRUE
            Textfield (15,30 350x30), "Threshold Editable"
            Checkbox (380,72 30x30), "Checkbox", variable: DALI_Commissioning.fbPart208Switching.bAddressingPhysical, input disabled if: TRUE
    Textfield (50,400 355x30), "Addressing Per Physical Selection Supported"
    Button (410,515 150x40), "Read"
        OnMouseClick: execute { DALI_Commissioning.fbPart208Switching.bRead := TRUE; }
    Button (580,515 150x40), "Write"
        OnMouseClick: execute { DALI_Commissioning.fbPart208Switching.bWrite := TRUE; }
    WaitingSymbolFlower (370,200 70x70), invisible if: DALI_Commissioning.fbPart208Switching.bHideWaitSymbol
    Button (285,90 50x30), "%d", text variable: DALI_Commissioning.fbPart208Switching.nUpSwitchOnThreshold
        OnMouseClick: write the text variable via Default, min 0, max 255, title "Up Switch On Threshold"
    Button (285,130 50x30), "%d", text variable: DALI_Commissioning.fbPart208Switching.nUpSwitchOffThreshold
        OnMouseClick: write the text variable via Default, min 0, max 255, title "Up Switch Off Threshold"
    Button (285,170 50x30), "%d", text variable: DALI_Commissioning.fbPart208Switching.nDownSwitchOnThreshold
        OnMouseClick: write the text variable via Default, min 0, max 255, title "Down Switch On Threshold"
    Button (285,210 50x30), "%d", text variable: DALI_Commissioning.fbPart208Switching.nDownSwitchOffThreshold
        OnMouseClick: write the text variable via Default, min 0, max 255, title "Down Switch Off Threshold"
END_VISUALIZATION

// ---- POUs/DALI/DALI_Setup/VISUs/Visu_DALICommissioning/Visu_Part300GenericDevice.TcVIS
